Omron CX-Programmer project 新工程 (CX-Programmer 9.61)

# PLC 后氦检2: CJ2M CPU33
I/O table (CPU CJ2M-CPU33): rack 0 slot 0 CJ1W-SCU21-V1; rack 0 slot 1 CJ1W-AD041-V1; rack 0 slot 2 CJ1W-ID261; rack 0 slot 3 CJ1W-OD231; rack 0 slot 4 CJ1W-OC201; rack 0 slot 11 CJ2M-EIP21

## Global symbols (name address type ; comment)
0.00 BOOL  ; 外来拉有料感应1
0.01 BOOL  ; 上料有料感应
0.02 BOOL  ; 电池跟随检测
0.03 BOOL  ; 扫码位有料感应
0.04 BOOL  ; 上料位柔性报警（常闭）
0.05 BOOL  ; 上料提升气缸原位
0.06 BOOL  ; 上料提升气缸到位
0.07 BOOL  ; 上料升降气缸原位
0.08 BOOL  ; 上料升降气缸到位(右）
0.09 BOOL  ; 右升降缸原位
0.10 BOOL  ; 右升降缸到位
0.11 BOOL  ; 上料左夹爪张开位
0.12 BOOL  ; 上料左夹爪夹紧位
0.13 BOOL  ; 上料右夹爪张开位
0.14 BOOL  ; 上料右夹爪夹紧位
0.15 BOOL  ; #1氦检阀原位
100.04 BOOL  ; 报警清除
101.00 BOOL  ; 手动放料限制条件
101.01 BOOL  ; 上料手动放料条件
102.00 BOOL  ; 放料停止拉带
110.00 BOOL  ; 整机复位按钮(T)
11.05 BOOL  ; #1腔体氦检阀
12.00 BOOL  ; #2腔体氦检阀
12.11 BOOL  ; #3腔体氦检阀
131.04 BOOL  ; 左扫码(M)
13.06 BOOL  ; #4腔体氦检阀
1534.15 BOOL  ; 单元1的串口1协议宏执行标志
1544.15 BOOL  ; 单元1串口2协议执行标志
1550.03 BOOL  ; 单元2串口1异常退出
1559.15 BOOL  ; 单元2串口1协议宏执行标志
1584.15 BOOL  ; SCU21_3 Port#1 Protocol Macro Executing Flag
15.05 BOOL  ; --
1600.03 BOOL  ; SCU21_4 Port#1 Abort Switch
1609.15 BOOL  ; SCU21_4 Port#1 Protocol Macro Executing Flag
16.00 BOOL  ; 故障计时按钮
16.01 BOOL  ; 故障计时清空按钮
1.00 BOOL  ; #2氦检阀原位
1.01 BOOL  ; 氦检1合模气缸原位
1.02 BOOL  ; 氦检1合模气缸到位
1.03 BOOL  ; 氦检2合模气缸原位
1.04 BOOL  ; 氦检2合模气缸到位
1.05 BOOL  ; 下料提升气缸原位
1.06 BOOL  ; 下料提升气缸到位
1.07 BOOL  ; 进料扫码阻挡缩回
1.08 BOOL  ; 进料扫码阻挡伸出
1.09 BOOL  ; 下料左夹爪张开位
1.10 BOOL  ; 下料左夹爪夹紧位
1.11 BOOL  ; 下料右夹爪张开位
1.12 BOOL  ; 下料右夹爪夹紧位
1.13 BOOL  ; 可出料信号
1.14 BOOL  ; 内部机台对接（下机台输出信号7.01）
1.15 BOOL  ; 下料位有料感应3
2000 CHANNEL  ; #1真空计度读出值CHO
2001 CHANNEL  ; #1真空计读出值CH1
2002 CHANNEL  ; #2真空计读出值CH2
2029.00 BOOL  ; #1真空计断线
2029.01 BOOL  ; #2真空计断线
20.00 BOOL  ; 自动模式切换按钮(T)
20.01 BOOL  ; 自动启动按钮(T)
20.02 BOOL  ; 自动停止按钮(T)
20.06 BOOL  ; 氦检仪内部校准
20.07 BOOL  ; 柔性报警解除按钮(T)
20.12 BOOL  ; 氦检仪内部校准
2906.06 BOOL  ; 进料机械手左极限
2906.07 BOOL  ; 进料机械手右极限
2906.08 BOOL  ; 出料机械手左极限
2906.09 BOOL  ; 出料机械手右极限
2960.00 BOOL  ; 上料伺服原点
2960.01 BOOL  ; 上料伺服近原点
2960.02 BOOL  ; 下料伺服原点
2960.03 BOOL  ; 下料伺服近原点
2960.04 BOOL  ; 备用
2960.05 BOOL  ; 备用
2960.06 BOOL  ; 上料伺负向限位
2960.07 BOOL  ; 上料伺服正向限位
2960.08 BOOL  ; 下料伺服负方向限位
2960.09 BOOL  ; 下料伺服正方向限位
2961.00 BOOL  ; 上料伺服脉冲
2961.01 BOOL  ; 下料伺服脉冲
2961.02 BOOL  ; 上料伺服方向
2961.03 BOOL  ; 下料伺服方向
2961.04 BOOL  ; 下一机台故障时，控制下一机台出料输送带（接到下一台机的7.15同一电机）
2.00 BOOL  ; 氦检仪报警信号
2.01 BOOL  ; 内部机台对接信号（后面一台后氦检下料位有料感应，即3。01）
2.02 BOOL  ; 内部机台对接（后面一台后氦检的出料拉带末端有料感应，即3.03）
2.03 BOOL  ; 下料柔性报警（常闭）
2.04 BOOL  ; 气源压力信号
2.05 BOOL  ; 上料伺服准备好
2.06 BOOL  ; 下料伺服准备好
2.07 BOOL  ; 上料伺服报警
2.08 BOOL  ; 下料伺服报警
2.09 BOOL  ; NG气缸原位
2.10 BOOL  ; NG气缸到位
2.11 BOOL  ; 扫码NG缸原位
2.12 BOOL  ; 扫码NG缸到位
2.13 BOOL  ; 扫码NG放料位有料感应
2.14 BOOL  ; 扫码NG槽溢出
2.15 BOOL  ; 扫码NG放料位有料感应
31.04 BOOL  ; #1电池扫码按钮
3.00 BOOL  ; 下料位光栅感应(常闭)
3.01 BOOL  ; 腔体1有料
3.02 BOOL  ; 下料位有料感应(常闭)
3.03 BOOL  ; 下料拉带末端有料感应(常闭)
3.04 BOOL  ; NG溢出感应
3.05 BOOL  ; 真空泵缺相
3.06 BOOL  ; 腔体2有料
3.07 BOOL  ; 过渡拉带末端有料感应
3.08 BOOL  ; 启动按钮
3.09 BOOL  ; 停止按钮
3.10 BOOL  ; 复位按钮
3.11 BOOL  ; 急停按钮
3.12 BOOL  ; 前门禁信号
3.13 BOOL  ; 后门禁信号
3.14 BOOL  ; 左门禁信号
3.15 BOOL  ; 右门禁信号
52.00 BOOL  ; 全部清零按钮
52.02 BOOL  ; OK数清零按钮
52.04 BOOL  ; NG数清零按钮
6.00 BOOL  ; 上料提升气缸
6.01 BOOL  ; #1上料升降气缸（左）
6.02 BOOL  ; #2上料升降气缸（右）
6.03 BOOL  ; 上料左夹爪
6.04 BOOL  ; 上料右夹爪
6.05 BOOL  ; 氦检1合模气缸伸出 关腔体
6.06 BOOL  ; 氦检1合模气缸缩回 开腔体
6.07 BOOL  ; 氦检2合模气缸伸出
6.08 BOOL  ; 氦检2合模气缸缩回
6.09 BOOL  ; 氦检1抽真空阀
6.10 BOOL  ; 氦检1氦检阀
6.11 BOOL  ; 氦检1破真空阀
6.12 BOOL  ; 氦检1吹气阀
6.13 BOOL  ; 氦检2抽真空
6.14 BOOL  ; 氦检2氦检阀
6.15 BOOL  ; 氦检2破真空阀
782 CHANNEL  ; 校验通信异常延时
7.00 BOOL  ; 氦检2吹气阀
7.01 BOOL  ; 内部机台对接（本机台给上机台信号1.14）
7.02 BOOL  ; 扫码阻挡气缸
7.03 BOOL  ; 上料私服使能
7.04 BOOL  ; 下料私服使能
7.05 BOOL  ; 过渡拉带启动
7.06 BOOL  ; 氦检仪电源开启
7.07 BOOL  ; 氦检仪启动
7.08 BOOL  ; 下料提升气缸
7.09 BOOL  ; 上工站可往下放料信号
7.10 BOOL  ; 下料左夹爪
7.11 BOOL  ; 下料右夹爪
7.12 BOOL  ; NG气缸
7.13 BOOL  ; 扫码NG缸
7.14 BOOL  ; 进料输送带电机
7.15 BOOL  ; 出料输送带电机
8.00 BOOL  ; 启动指示灯
8.01 BOOL  ; 停止指示灯
8.02 BOOL  ; 复位指示灯
8.03 BOOL  ; 三色灯-红
8.04 BOOL  ; 三色灯-绿
8.05 BOOL  ; 三色灯-黄
8.06 BOOL  ; 蜂鸣器
8.07 BOOL  ; 真空泵
9.04 BOOL  ; 氦检电源打开
A202.01 BOOL  ; 通信端口1允许标志
A202.02 BOOL  ; 通信端口2允许标志
A202.03 BOOL  ; 通信端口3允许标志
A276 CHANNEL  ; 前机械手当前脉冲
A278 CHANNEL  ; 下料机械手当前脉冲
A280.04 BOOL  ; 上料机械手脉冲输出中
A280.05 BOOL  ; 上料轴无原点标志
A281.04 BOOL  ; 下料机械手脉冲输出中
A281.05 BOOL  ; 下料轴无原点标志
A322 CHANNEL  ; 进料旋转当前位置脉冲
A324 CHANNEL  ; 出料旋转当前位置脉冲
A326.04 BOOL  ; 进料旋转脉冲输出中
A326.05 BOOL  ; 上料旋转原点标志
A327.04 BOOL  ; 出料旋转脉冲输出中
A327.05 BOOL  ; 下料旋转原点标志
A351 CHANNEL  ; 系统时间
A540.08 BOOL  ; 上料机械手CW
A540.09 BOOL  ; 上料机械手CCW
A541.08 BOOL  ; 下料机械手CW
A541.09 BOOL  ; 下料机械手CCW
A542.08 BOOL  ; 进料旋转CCW
A542.09 BOOL  ; 进料旋转CW
A543.08 BOOL  ; 出料旋转CCW
A543.09 BOOL  ; 出料旋转CW
D0 CHANNEL  ; 上料机械手自动速度mm/s
D10 CHANNEL  ; 上料左夹位
D100 CHANNEL  ; 外来拉有料感应1延时HMI
D1000 CHANNEL  ; #1腔体检漏口压力(浮点)
D1002 CHANNEL  ; #1腔体漏率(浮点)
D1004 CHANNEL  ; #1腔体测试完成时的检漏口压力
D1006 CHANNEL  ; #1腔体测试完成时的漏率
D101 CHANNEL  ; 外来拉有料感应2延时HMI
D102 CHANNEL  ; 上料位有料感应延时HMI
D1020 CHANNEL  ; #2腔体检漏口压力(浮点)
D1022 CHANNEL  ; #2腔体漏率(浮点)
D1024 CHANNEL  ; #2腔体测试完成时检漏口压力
D1026 CHANNEL  ; #2腔体测试完成时的漏率
D103 CHANNEL  ; 上料位有料感应2延时HMI
D104 CHANNEL  ; 上料位柔性报警（常闭）延时
D105 CHANNEL  ; 上料提升气缸原位延时
D106 CHANNEL  ; 上料提升气缸到位延时
D107 CHANNEL  ; 上料升降气缸原位延时
D108 CHANNEL  ; 上料升降气缸到位延时
D109 CHANNEL  ; 扫码阻挡气缸原位延时
D110 CHANNEL  ; 扫码阻挡气缸到位延时
D1100 CHANNEL  ; 测试
D111 CHANNEL  ; 上料左夹爪张开位延时
D112 CHANNEL  ; 上料左夹爪夹紧位延时
D113 CHANNEL  ; 上料右夹爪张开位延时
D114 CHANNEL  ; 上料右夹爪夹紧位延时
D1140 CHANNEL  ; HMI 页面
D115 CHANNEL  ; #1氦检阀原位延时时间
D116 CHANNEL  ; #2氦检阀原位延时时间
D117 CHANNEL  ; 氦检1合模气缸原位延时
D118 CHANNEL  ; 氦检1合模气缸到位延时
D119 CHANNEL  ; 氦检2合模气缸原位延时
D12 CHANNEL  ; 下料右夹爪OK放料位
D120 CHANNEL  ; 氦检2合模气缸到位延时
D1204 CHANNEL  ; 检漏口压力设定值
D1206 CHANNEL  ; 漏率设定值
D121 CHANNEL  ; 下料提升气缸原位延时
D1210 CHANNEL  ; 氦检仪稳定设定时间
D122 CHANNEL  ; 下料提升气缸到位延时
D123 CHANNEL  ; 下料升降气缸原位延时
D124 CHANNEL  ; 下料升降气缸到位延时
D125 CHANNEL  ; 下料左夹爪张开位延时
D1250 CHANNEL  ; 检漏口压力设定值小数部分
D1252 CHANNEL  ; 检漏口压力设定值指数
D1254 CHANNEL  ; 漏率设定值小数部分
D1256 CHANNEL  ; 漏率设定值指数
D126 CHANNEL  ; 下料左夹爪夹紧位延时
D1260 CHANNEL  ; 检漏口压力底数转换
D1264 CHANNEL  ; 漏率底数转换
D1266 CHANNEL  ; 漏率设定值(浮点数Pa.m3)
D127 CHANNEL  ; 下料右夹爪张开位延时
D1270 CHANNEL  ; 注氦嘴气密性设定值小数部分
D1272 CHANNEL  ; 注氦嘴气密性设定值指数
D1274 CHANNEL  ; 注氦嘴气密性设定值指数部分
D1276 CHANNEL  ; 注氦嘴气密性设定值(Float)
D1278 CHANNEL  ; 清氦次数设定值
D128 CHANNEL  ; 下料右夹爪夹紧位延时
D129 CHANNEL  ; 备用
D130 CHANNEL  ; 备用
D131 CHANNEL  ; 备用
D1310 CHANNEL  ; 氦检仪稳定漏率设定值小数
D1312 CHANNEL  ; 氦检仪稳定漏率设定值指数
D1316 CHANNEL  ; 氦检仪稳定漏率设定值(Float)
D132 CHANNEL  ; 氦检仪报警信号延时
D133 CHANNEL  ; 备用
D134 CHANNEL  ; 备用
D135 CHANNEL  ; 下料柔性报警（常闭）延时
D136 CHANNEL  ; 气源压力信号延时
D137 CHANNEL  ; 上料伺服准备好延时
D138 CHANNEL  ; 下料伺服准备好延时
D139 CHANNEL  ; 备用
D140 CHANNEL  ; 备用
D141 CHANNEL  ; NG气缸原位延时
D1416 CHANNEL  ; 氦检仪压力异常延时
D142 CHANNEL  ; NG气缸到位延时
D143 CHANNEL  ; 工站给予信号时间
D144 CHANNEL  ; 扫码NG缸原位时间
D145 CHANNEL  ; 扫码NG缸原位时间
D146 CHANNEL  ; 备用
D147 CHANNEL  ; 备用
D148 CHANNEL  ; 1#腔体有料延时
D149 CHANNEL  ; 2#腔体有料延时
D150 CHANNEL  ; 下料位有料感应1延时
D151 CHANNEL  ; 下料位有料感应2延时
D152 CHANNEL  ; NG溢出感应延时
D153 CHANNEL  ; 真空泵缺相延时
D154 CHANNEL  ; 备用
D155 CHANNEL  ; 备用
D156 CHANNEL  ; 启动按钮延时
D157 CHANNEL  ; 停止按钮延时
D158 CHANNEL  ; 复位按钮延时
D159 CHANNEL  ; 急停按钮延时
D1590 CHANNEL  ; 扫码位暂存码1
D16 CHANNEL  ; 上料左扫码NG参数
D160 CHANNEL  ; 前门禁信号延时
D1600 CHANNEL  ; 扫码位暂存码
D161 CHANNEL  ; 后门禁信号延时
D162 CHANNEL  ; 左门禁信号延时
D163 CHANNEL  ; 右门禁信号延时
D168 CHANNEL  ; 传感器延迟时间
D1790 CHANNEL  ; 上料位待料延时设定HMI
D18 CHANNEL  ; 上料右扫码NG参数
D180 CHANNEL  ; 上料机械手当前脉冲
D1802 CHANNEL  ; TS
D182 CHANNEL  ; 上料机械手当前脉冲(浮点)
D184 CHANNEL  ; 伺服脉冲当量(浮点)
D1840 CHANNEL  ; 下料右爪测试检漏口压力结果
D1842 CHANNEL  ; 下料右爪测试漏率结果
D1844 CHANNEL  ; 下料右爪 测试结果
D1846 CHANNEL  ; 下料左爪压力
D1848 CHANNEL  ; 下料左爪漏率
D1850 CHANNEL  ; 下料左爪测试结果
D1858 CHANNEL  ; 下料右爪测试检漏口压力结果PC
D186 CHANNEL  ; 上料机械手当前位置(mm)
D1860 CHANNEL  ; 下料右爪测试漏率结果PC
D1862 CHANNEL  ; 下料右爪 测试结果pC
D1868 CHANNEL  ; 下料左爪压力PC
D1870 CHANNEL  ; 下料左爪漏率PC
D1872 CHANNEL  ; 下料左爪测试结果PC
D188 CHANNEL  ; 伺服脉冲当量
D1880 CHANNEL  ; 1爪腔体编号
D1881 CHANNEL  ; 2爪腔体编号
D190 CHANNEL  ; 下料机械手当前脉冲
D1900 CHANNEL  ; 下料右爪电池工位PC
D1901 CHANNEL  ; 传输完成地址
D1902 CHANNEL  ; 下料左爪工位PC
D1903 CHANNEL  ; 传输完成-左
D1904 CHANNEL  ; 传输完成地址
D1905 CHANNEL  ; 传输完成-左
D192 CHANNEL  ; 下料机械手当前脉冲(浮点)
D196 CHANNEL  ; 下料机械手当前位置(mm)
D198 CHANNEL  ; 上下料机械手距各自原点的总距离
D2 CHANNEL  ; 上料机械手手动速度mm/s
D20 CHANNEL  ; 下料机械手自动速度mm/s
D200 CHANNEL  ; #1腔体真空值
D2000 CHANNEL  ; 氦检仪当前实时漏率
D20000 CHANNEL  ; #1,#2路模拟量使用设置
D20001 CHANNEL  ; #1,#2路模拟量输入范围位0--10v
D20018 CHANNEL  ; #1,#2路模拟量分辨率8000，普通模式
D210 CHANNEL  ; #2腔体真空值
D22 CHANNEL  ; 下料机械手动速度mm/s
D230 CHANNEL  ; #1腔体抽气时间
D232 CHANNEL  ; #2腔体抽气时间
D234 CHANNEL  ; 1屏蔽2带料3测试中4测试完成
D236 CHANNEL  ; 1屏蔽2带料3测试中4测试完成
D238 CHANNEL  ; #1腔体测试结果
D239 CHANNEL  ; #2腔体测试结果
D24 CHANNEL  ; 下料机械手腔体1位置(mm)
D240 CHANNEL  ; 接收检漏仪状态的起始字
D241 CHANNEL  ; 接收的检漏口压力(ASCII)
D2450 CHANNEL  ; 氦捡仪稳定时间设定值(BCD)
D2452 CHANNEL  ; #1氦检阀打开抽气阀关闭延时
D2454 CHANNEL  ; #2氦检阀打开抽气阀关闭延时
D2456 CHANNEL  ; 氦检关真空延时
D250 CHANNEL  ; 接收检漏口压力的起始字
D251 CHANNEL  ; 接收的检漏口压力(ASCII)
D26 CHANNEL  ; 下料机械手腔体2位置(mm)
D260 CHANNEL  ; 接收漏率起始字
D261 CHANNEL  ; 接收的漏率(ASCII)
D270 CHANNEL  ; 上下料机械手原点间距离
D272 CHANNEL  ; 机械手治具宽度
D274 CHANNEL  ; 上下料机械手间的距离
D28 CHANNEL  ; 下料机械手左夹爪OK放料位置(mm)
D282 CHANNEL  ; .
D290 CHANNEL  ; 180浮点数
D294 CHANNEL  ; 180度脉冲数
D298 CHANNEL  ; 进料位置+180度角
D30 CHANNEL  ; 下料机械手NG放料位置(mm)
D300 CHANNEL  ; 外来拉有料感应1延时
D301 CHANNEL  ; 外来料感应2
D302 CHANNEL  ; 上料位有料感应1
D303 CHANNEL  ; 上料位有料延时
D304 CHANNEL  ; 柔性报警
D3040 CHANNEL  ; 取料位条码
D305 CHANNEL  ; 上料提升原位延时
D306 CHANNEL  ; 上料提升延时
D3060 CHANNEL  ; 右夹子条码
D307 CHANNEL  ; 上料升降延时
D308 CHANNEL  ; 上料升降到位延时
D3080 CHANNEL  ; 上料左夹子条码
D309 CHANNEL  ; 右升降原位延时间
D310 CHANNEL  ; 右升降缸到位时间
D3100 CHANNEL  ; 腔体1右待测料条码
D311 CHANNEL  ; 上左爪张开位
D312 CHANNEL  ; 上左夹紧延时
D3120 CHANNEL  ; 腔体2左位条码
D313 CHANNEL  ; 上右爪松开延时
D314 CHANNEL  ; 上右夹紧延时
D3140 CHANNEL  ; 腔体2右位条码
D3160 CHANNEL  ; 腔体1左待测条码
D317 CHANNEL  ; 合模1原位延时
D318 CHANNEL  ; 合模1到位延时
D3180 CHANNEL  ; 下料右爪条码
D319 CHANNEL  ; 合模2原位延时
D32 CHANNEL  ; 出料旋转步进自动速度(度/s）
D320 CHANNEL  ; 合模2到位延时
D3200 CHANNEL  ; 下料左爪条码
D321 CHANNEL  ; 下料提升原位延时
D322 CHANNEL  ; 下料提升到位延时
D3220 CHANNEL  ; 下料右爪条码PC
D323 CHANNEL  ; 备用
D324 CHANNEL  ; 备用
D3240 CHANNEL  ; 下料左爪条码PC
D325 CHANNEL  ; 下左爪张开延时
D326 CHANNEL  ; 下左夹紧延时
D327 CHANNEL  ; 下右爪张开位延时
D328 CHANNEL  ; 下右爪夹紧位延时
D332 CHANNEL  ; 氦检报警延时
D335 CHANNEL  ; 下料柔性报警延时
D336 CHANNEL  ; 气压报警延时
D34 CHANNEL  ; 出料旋转步进手动速度(度/s)
D341 CHANNEL  ; NG气缸原位延时
D342 CHANNEL  ; NG气缸到位延时
D348 CHANNEL  ; 1#腔体有料延时
D349 CHANNEL  ; 2#腔体有料延时
D350 CHANNEL  ; 下料位有料感应1延时
D351 CHANNEL  ; 下料位有料感应2延时
D353 CHANNEL  ; 真空泵缺相
D36 CHANNEL  ; 出料旋转步进出料角度1(mm)
D370 CHANNEL  ; 氦检仪就绪状态
D38 CHANNEL  ; 出料旋转步进下料角度
D4 CHANNEL  ; 上料机械手右夹爪位(浮点)
D40 CHANNEL  ; 腔体真空达到阀值
D400 CHANNEL  ; 上料机械手自动状态加速度
D4000 CHANNEL  ; 真空值1转存
D4002 CHANNEL  ; #1真空值运算1
D4004 CHANNEL  ; #1真空值运算2
D4006 CHANNEL  ; #1真空值运算3
D4008 CHANNEL  ; #1真空值运算4
D401 CHANNEL  ; 上料机械手自动状态减速度
D4010 CHANNEL  ; 腔体1实际真空值(浮点)
D402 CHANNEL  ; 上料机械手自动速度puls/s
D4020 CHANNEL  ; 真空值2转存
D4022 CHANNEL  ; #2真空值运算1
D4024 CHANNEL  ; #2真空值运算2
D4026 CHANNEL  ; #2真空值运算3
D4028 CHANNEL  ; #2真空值运算4
D404 CHANNEL  ; 上料机械手自动位移量
D406 CHANNEL  ; 上料机械手自动状态起动速度
D410 CHANNEL  ; 上料机械手手动状态加速度
D411 CHANNEL  ; 上料机械手手动状态减速度
D412 CHANNEL  ; 上料机械手手动速度puls/s
D414 CHANNEL  ; 上料机械手手动位移量
D416 CHANNEL  ; 上料机械手手动状态起动速度
D42 CHANNEL  ; 腔体抽气时间
D420 CHANNEL  ; 下料机械手自动状态加速度
D421 CHANNEL  ; 下料机械手自动状态减速度
D422 CHANNEL  ; 下料机械手自动速度puls/s
D424 CHANNEL  ; 下料机械手自动位移量
D426 CHANNEL  ; 下料机械手自动状体起动速度
D430 CHANNEL  ; 下料机械手手动状态加速度
D431 CHANNEL  ; 下料机械手手动状态减速度
D432 CHANNEL  ; 下料机械手手动速度puls/s
D434 CHANNEL  ; 下料机械手手动位移量
D436 CHANNEL  ; 下料机械手手动状态起动速度
D44 CHANNEL  ; 抽残气后压力设置值
D440 CHANNEL  ; 进料旋转步进自动状态加速度
D441 CHANNEL  ; 进料旋转步进自动状体减速度
D442 CHANNEL  ; 进料旋转步进自动速度puls/s
D444 CHANNEL  ; 进料旋转自动位移量
D446 CHANNEL  ; 进料旋转步进自动状态起动速度
D450 CHANNEL  ; 进料旋转步进手动状态加速度
D451 CHANNEL  ; 进料旋转步进手动状态减速度
D452 CHANNEL  ; 进料旋转步进手动速度puls/s
D456 CHANNEL  ; 进料旋转步进手动状态起动速度
D46 CHANNEL  ; 氦检设定时间
D460 CHANNEL  ; 出料旋转步进自动状态加速度
D461 CHANNEL  ; 出料旋转步进自动状态减速度
D462 CHANNEL  ; 出料旋转步进自动速度puls/s
D464 CHANNEL  ; 出料旋转自动位移量
D466 CHANNEL  ; 出料旋转步进自动状态起动速度
D470 CHANNEL  ; 出料旋转步进手动状态加速度
D471 CHANNEL  ; 出料旋转步进手动状态减速度
D472 CHANNEL  ; 出料旋转步进手动速度puls/s
D476 CHANNEL  ; 出料旋转步进手动状态起动速度
D48 CHANNEL  ; 腔体破真空设定值
D480 CHANNEL  ; 上下料机械手正向行程脉冲
D484 CHANNEL  ; 上下料机械手反向行程
D488 CHANNEL  ; 上下料机械手反向行程脉冲
D50 CHANNEL  ; 检漏口压力指数
D500 CHANNEL  ; 上料机械手自动速度puls/s
D5000 CHANNEL  ; 扫码1长度
D504 CHANNEL  ; 上料机械手手动速度puls/s
D510 CHANNEL  ; 下料机械手自动速度puls/s
D514 CHANNEL  ; 下料机械手手动速度puls/s
D5198 CHANNEL  ; 流入个数
D52 CHANNEL  ; 检漏口压力底数
D520 CHANNEL  ; 进料旋转步进自动速度puls/s
D5200 CHANNEL  ; 流出个数
D5202 CHANNEL  ; OK个数
D5204 CHANNEL  ; 检测NG个数
D5206 CHANNEL  ; 良率
D5220 CHANNEL  ; 扫码NG个数
D5222 CHANNEL  ; 检测产量
D524 CHANNEL  ; 进料旋转步进手动速度puls/s
D530 CHANNEL  ; 出料旋转步进自动速度puls/s
D534 CHANNEL  ; 出料旋转步进手动速度puls/s
D54 CHANNEL  ; 漏率指数
D5430 CHANNEL  ; PPM统计
D5432 CHANNEL  ; 下料数量
D5434 CHANNEL  ; 计时
D550 CHANNEL  ; 上料机械手在（右）扫码NG位..
D552 CHANNEL  ; 上料机械手在（左）NG槽参数
D56 CHANNEL  ; 漏率底数
D580 CHANNEL  ; 下料右爪放OK料位置（浮点）
D584 CHANNEL  ; 下料右爪放OK料位置脉冲
D592 CHANNEL  ; 上料机械手左夹爪位置脉冲(浮点)
D596 CHANNEL  ; 上料机械手左夹爪位置脉冲
D6 CHANNEL  ; 上料机械手腔体1位置(浮点)
D60 CHANNEL  ; 腔体自检真空阀值
D600 CHANNEL  ; 上料机械手右夹爪位置脉冲(浮点)
D602 CHANNEL  ; 氦检上限位值
D604 CHANNEL  ; 上料机械手右夹爪位置脉冲
D610 CHANNEL  ; 上料机械手腔体1位置脉冲(浮点)
D6100 CHANNEL  ; 2个电芯出料计时
D614 CHANNEL  ; 上料机械手腔体1位置脉冲
D62 CHANNEL  ; 腔体自检抽气时间
D620 CHANNEL  ; 上料机械手腔体2位置(浮点)
D6200 CHANNEL  ; 2个电芯生产周期
D624 CHANNEL  ; 上料机械手腔体2位置脉冲
D626 CHANNEL  ; 上料机械手在（右）扫码NG位
D628 CHANNEL  ; 上料机械手在（左）NG槽参数
D630 CHANNEL  ; 下料机械手腔体1位置(浮点)
D6300 CHANNEL  ; PPM
D634 CHANNEL  ; 下料机械手腔体1位置脉冲
D64 CHANNEL  ; 腔体自检泄漏量设置值
D640 CHANNEL  ; 下料机械手腔体2位置(浮点)
D644 CHANNEL  ; 下料机械手腔体2位置脉冲
D650 CHANNEL  ; 下料机械手左爪OK放料位置(浮点)
D654 CHANNEL  ; 下料机械手左爪OK放料位置脉冲
D66 CHANNEL  ; 条码设置长度
D660 CHANNEL  ; 下料机械手NG放料位置(浮点)
D664 CHANNEL  ; 下料机械手NG放料位置脉冲
D670 CHANNEL  ; 氦检下限位值
D672 CHANNEL  ; 氦检上限位值
D674 CHANNEL  ; 进料旋转进料位置1脉冲
D68 CHANNEL  ; 腔体自检保压前设定时间
D680 CHANNEL  ; 进料旋转上料位置(浮点)
D684 CHANNEL  ; 进料旋转上料位置脉冲
D688 CHANNEL  ; 进料旋转上料位置+180度位置脉冲
D690 CHANNEL  ; 出料旋转出料位置1(浮点)
D694 CHANNEL  ; 出料旋转出料位置1脉冲
D70 CHANNEL  ; 腔体自检保压设定时间
D700 CHANNEL  ; 出料旋转下料位置(浮点)
D7000 CHANNEL  ; #1扫码长度
D7001 CHANNEL  ; #1电池条码
D704 CHANNEL  ; 出料旋转下料位置脉冲
D710 CHANNEL  ; 旋转步进正向行程脉冲
D714 CHANNEL  ; 旋转步进反向行程
D72 CHANNEL  ; 腔体自检破真空设定值
D720 CHANNEL  ; 轴控制预留
D734 CHANNEL  ; 旋转步进反向行程脉冲
D74 CHANNEL  ; #1腔体保压前真空值
D76 CHANNEL  ; #1腔体保压后真空值
D78 CHANNEL  ; #1腔体自检泄漏量
D780 CHANNEL  ; 进料旋转步进进料角度2(mm)
D782 CHANNEL  ; 进料旋转进料位置2(浮点)
D784 CHANNEL  ; 进料旋转进料位置2脉冲
D792 CHANNEL  ; 出料旋转出料位置2(浮点)
D794 CHANNEL  ; 出料旋转出料位置2脉冲
D8 CHANNEL  ; 上料机械手腔体2位置(浮点)
D80 CHANNEL  ; #2腔体保压前真空值
D800 CHANNEL  ; 氦检时间(储存)
D8000 CHANNEL  ; 检漏状态第一字节
D8001 CHANNEL  ; 检漏状态第二字节
D8002 CHANNEL  ; 检漏状态结束字节
D8010 CHANNEL  ; 待机状态第一字节
D8011 CHANNEL  ; 待机状态第二字节
D8012 CHANNEL  ; 待机状态结束字节
D802 CHANNEL  ; 检漏口压力指数(储存)
D8020 CHANNEL  ; 定标状态第一字节
D8021 CHANNEL  ; 定标状态第二字节
D8022 CHANNEL  ; 定标状态结束字节
D8030 CHANNEL  ; 启动状态第一字节
D8031 CHANNEL  ; 启动状态第二字节
D8032 CHANNEL  ; 启动状态结束字节
D804 CHANNEL  ; 检漏口压力底数(储存)
D8040 CHANNEL  ; 错误状态第一字节
D8041 CHANNEL  ; 错误状态第二字节
D8042 CHANNEL  ; 错误状态结束字节
D8050 CHANNEL  ; 暂停状态第一字节
D8051 CHANNEL  ; 暂停状态第二字节
D8052 CHANNEL  ; 暂停状态结束字节
D806 CHANNEL  ; 漏率指数
D808 CHANNEL  ; 漏率底数
D8100 CHANNEL  ; 氦检仪状态(1-检漏,2-待机,3-启动,4-定标,5-错误,6-暂停)
D82 CHANNEL  ; #1腔体保压后真空值
D820 CHANNEL  ; 设备状态
D821 CHANNEL  ; 设备状态(储存)
D822 CHANNEL  ; 设备状态变更
D830 CHANNEL  ; 早班分、秒
D8300 CHANNEL  ; 校验触发
D8302 CHANNEL  ; 校验结果（1-OK，2-NG）
D831 CHANNEL  ; 早班日、时
D832 CHANNEL  ; 晚班分、秒
D833 CHANNEL  ; 晚班分、秒
D834 CHANNEL  ; 晚班日、时
D836 CHANNEL  ; 只比较时、分、秒
D838 CHANNEL  ; 晚班传输信号
D84 CHANNEL  ; #2腔体自检泄漏量
D840 CHANNEL  ; 单班生产时间
D8400 CHANNEL  ; 读氦检仪报警
D842 CHANNEL  ; 单班故障时间
D8500 CHANNEL  ; 读氦检仪内部校准状态
D8600 CHANNEL  ; 氦检校准暂存状态1-完成
D8601 CHANNEL  ; 氦检校准暂存状态1-完成
D8610 CHANNEL  ; 氦检校准暂存状态2-通过
D8611 CHANNEL  ; 氦检校准暂存状态2-通过
D8612 CHANNEL  ; 氦检校准暂存状态3
D8620 CHANNEL  ; 氦检校准暂存状态3-进行
D8621 CHANNEL  ; 氦检校准暂存状态3-进行
D8622 CHANNEL  ; 氦检校准暂存状态3-进行
D90 CHANNEL  ; #1腔体手动抽气时间
D9000 CHANNEL  ; PC交换地址
D91 CHANNEL  ; #1腔体保压前时间
D9100 CHANNEL  ; 上下料机械手总距离
D9102 CHANNEL  ; 原点距离
D9104 CHANNEL  ; 2轴相距距离
D92 CHANNEL  ; #1腔体保压时间
D93 CHANNEL  ; #2腔体自检抽气时间
D9300 CHANNEL  ; 放料状态
D94 CHANNEL  ; #2腔体进入保压前时间
D95 CHANNEL  ; #2腔体保压时间
D9500 CHANNEL  ; #1放料电池条码
D9520 CHANNEL  ; #2放料电池条码
D9591 CHANNEL  ; #1放料电池条码
D9592 CHANNEL  ; #1放料电池条码
D9593 CHANNEL  ; #1放料电池条码
D9594 CHANNEL  ; #1放料电池条码
D9595 CHANNEL  ; #1放料电池条码
D9596 CHANNEL  ; #1放料电池条码
D9597 CHANNEL  ; #1放料电池条码
D9598 CHANNEL  ; #1放料电池条码
D9599 CHANNEL  ; #1放料电池条码
D9601 CHANNEL  ; #2放料电池条码
D9602 CHANNEL  ; #2放料电池条码
D9603 CHANNEL  ; #2放料电池条码
D9604 CHANNEL  ; #2放料电池条码
D9605 CHANNEL  ; #2放料电池条码
D9606 CHANNEL  ; #2放料电池条码
D9607 CHANNEL  ; #2放料电池条码
D9608 CHANNEL  ; #2放料电池条码
D9609 CHANNEL  ; #2放料电池条码
D9612 CHANNEL  ; 放料电池实际漏率
D9613 CHANNEL  ; 放料电池实际漏率
D9614 CHANNEL  ; 放料电池实际检漏口压力
D9615 CHANNEL  ; 放料电池实际检漏口压力
D9616 CHANNEL  ; 放料电池电池工位
D9617 CHANNEL  ; 放料电池电池工位
D9618 CHANNEL  ; 放料电池电池测试结果
D9619 CHANNEL  ; 放料电池电池测试结果
D9630 CHANNEL  ; 漏率设定值
D9631 CHANNEL  ; 漏率设定值
D9632 CHANNEL  ; 检漏口压力设定值
D9633 CHANNEL  ; 检漏口压力设定值
D9634 CHANNEL  ; 氦检时间设定值
D9635 CHANNEL  ; 氦检时间设定值
D9999 CHANNEL  ; 程序修改日期
H0.00 BOOL  ; #1腔体启用
H0.01 BOOL  ; #2腔体启用
H0.02 BOOL  ; 扫码屏蔽（1-屏蔽)
H0.03 BOOL  ; 电脑屏蔽
H0.04 BOOL  ; 门磁开关启用
H0.05 BOOL  ; 0-正常程序/1-空跑程序
H0.06 BOOL  ; 氦检仪屏蔽
H0.07 BOOL  ; 重复扫码禁用
H0.08 BOOL  ; 真空屏蔽
H0.09 BOOL  ; 入料拉带停止选择
H10.00 BOOL  ; 夹爪下料区有电池
H110.00 BOOL  ; 新复位方式启用
H11.00 BOOL  ; 上料机械手归零完成
H16.02 BOOL  ; 下料夹爪1手动松开
H16.03 BOOL  ; 下料夹爪2手动松开
H16.04 BOOL  ; 下料夹爪3手动松开
H16.05 BOOL  ; 下料夹爪4手动松开
H1.00 BOOL  ; 外来拉有料感应1
H1.01 BOOL  ; 外来拉有料感应2(备用)
H1.02 BOOL  ; 上料位有料感应1
H1.03 BOOL  ; 上料位有料感应2
H1.04 BOOL  ; 上料位柔性报警（常闭）
H1.05 BOOL  ; 上料提升气缸原位
H1.06 BOOL  ; 上料提升气缸到位
H1.07 BOOL  ; 上料升降气缸原位
H1.08 BOOL  ; 上料升降气缸到位
H1.09 BOOL  ; 右升降缸原位屏蔽
H1.10 BOOL  ; 右升降缸到位屏蔽
H1.11 BOOL  ; 上料左夹爪张开位
H1.12 BOOL  ; 上料左夹爪夹紧位
H1.13 BOOL  ; 上料右夹爪张开位
H1.14 BOOL  ; 上料右夹爪夹紧位
H1.15 BOOL  ; #1氦检阀原位屏蔽
H2.00 BOOL  ; #2氦检阀原位屏蔽
H2.01 BOOL  ; 氦检1合模气缸原位
H2.02 BOOL  ; 氦检1合模气缸到位
H2.03 BOOL  ; 氦检2合模气缸原位
H2.04 BOOL  ; 氦检2合模气缸到位
H2.05 BOOL  ; 下料提升气缸原位
H2.06 BOOL  ; 下料提升气缸到位
H2.07 BOOL  ; 备用
H2.08 BOOL  ; 备用
H2.09 BOOL  ; 下料左夹爪张开位
H2.10 BOOL  ; 下料左夹爪夹紧位
H2.11 BOOL  ; 下料右夹爪张开位
H2.12 BOOL  ; 下料右夹爪夹紧位
H2.13 BOOL  ; 备用
H2.14 BOOL  ; 备用
H2.15 BOOL  ; 备用
H3.00 BOOL  ; 氦检仪报警信号
H3.01 BOOL  ; 备用
H3.02 BOOL  ; 备用
H3.03 BOOL  ; 下料柔性报警（常闭）
H3.04 BOOL  ; 气源压力信号
H3.05 BOOL  ; 上料伺服准备好
H3.06 BOOL  ; 下料伺服准备好
H3.07 BOOL  ; 备用
H3.08 BOOL  ; 备用
H3.09 BOOL  ; NG气缸原位
H3.10 BOOL  ; NG气缸到位
H3.11 BOOL  ; 下个工站给予信号
H3.12 BOOL  ; 扫码NG气缸原位屏蔽
H3.13 BOOL  ; 扫码NG气缸到位屏蔽
H3.14 BOOL  ; 备用
H3.15 BOOL  ; 备用
H40.02 BOOL  ; 扫码屏蔽-HMI
H40.07 BOOL  ; 扫码NG料（右）
H40.08 BOOL  ; 扫码NG（左）
H46.00 BOOL  ; 机台方向选择(0:左进右出,1:右进左出)
H4.00 BOOL  ; 1#腔体有料
H4.01 BOOL  ; 2#腔体有料
H4.02 BOOL  ; 下料位有料感应1
H4.03 BOOL  ; 下料位有料感应2
H4.04 BOOL  ; NG溢出感应
H4.05 BOOL  ; 真空泵缺相
H4.06 BOOL  ; 备用
H4.07 BOOL  ; 备用
H4.08 BOOL  ; 启动按钮
H4.09 BOOL  ; 停止按钮
H4.10 BOOL  ; 复位按钮
H4.11 BOOL  ; 急停按钮
H4.12 BOOL  ; 前门禁信号
H4.13 BOOL  ; 后门禁信号
H4.14 BOOL  ; 左门禁信号
H4.15 BOOL  ; 右门禁信号
H50 CHANNEL  ; 复位有料记忆
H50.00 BOOL  ; 扫码位有料
H50.01 BOOL  ; 上料左爪有料记忆
H50.02 BOOL  ; 上料右爪有料
H50.03 BOOL  ; 下料右爪有料
H50.04 BOOL  ; 下料右爪有料
H50.05 BOOL  ; 爪子无料
H50.06 BOOL  ; 上料位有料标志
H50.07 BOOL  ; 上右夹爪有料标志
H50.08 BOOL  ; 上左夹有料标志
H50.09 BOOL  ; #1腔体右位有待测料标志
H50.10 BOOL  ; #1腔体左位有料标志
H50.11 BOOL  ; 2号腔体右位有料标志
H50.12 BOOL  ; 2#腔体左位有料标志
H50.13 BOOL  ; #1腔体NG
H50.14 BOOL  ; #1腔体测试中
H51.00 BOOL  ; #1腔体测试结束
H51.01 BOOL  ; #2腔体测试结束
H51.02 BOOL  ; 下料左爪有料
H51.03 BOOL  ; 下料右爪有料标志
H51.04 BOOL  ; #2腔体放料完成
H51.05 BOOL  ; 腔体1放料完成标志
H51.06 BOOL  ; #2腔体产品NG
H51.07 BOOL  ; #2腔体测试中
H51.13 BOOL  ; 去腔体#2取料标志
H51.14 BOOL  ; 下料轴往1#取料标志
H53.00 BOOL  ; 上料轴归零完成
H53.01 BOOL  ; #1腔体自检泄露
H53.02 BOOL  ; #2腔体自检泄露
H54.00 BOOL  ; 下料轴归零完成
H55.00 BOOL  ; 上料轴往1#腔体放料标志
H55.01 BOOL  ; 上料轴往2#腔体放料标志
H56.00 BOOL  ; 跟随检测
H5.00 BOOL  ; 氦检仪屏蔽
H5.02 BOOL  ; 蜂鸣器屏蔽
H5.09 BOOL  ; MES采集漏率单位为mPa.m3/s(仪器显示值1000倍)
H60.09 BOOL  ; #1腔体右位有待测料
H60.10 BOOL  ; #1腔体左位有料标志
H60.11 BOOL  ; 2号腔体右位有料
H60.12 BOOL  ; 2#腔体左位有料
H6.00 BOOL  ; 机台方向选择(0:左进右出,1:右进左出)
H80.00 BOOL  ; 左爪手动记忆有料
H80.01 BOOL  ; 右爪手动记忆有料
H80.02 BOOL  ; 上料左爪手动记忆有料
H80.03 BOOL  ; 上料右爪手动记忆有料
H80.05 BOOL  ; 下料拉带2有料
H80.06 BOOL  ; 过渡拉带有料
H81.00 BOOL  ; 老氦检仪选择
H81.01 BOOL  ; 氦检仪电源打开—HMI
H9.00 BOOL  ; 单料模式
T0000 BOOL  ; 进料感应延时
T0001 BOOL  ; 上料柔性报警感应延时
T0002 BOOL  ; 下料柔性报警感应延时
T0003 BOOL  ; 出料柔性报警感应延时
T0004 BOOL  ; 气源压力信号感应延时
T0005 BOOL  ; 进料缓存有料信号延时
T0006 BOOL  ; 出料缓存有料信号延时
T0007 BOOL  ; 腔体有料信号
T0008 BOOL  ; 扫码缓存左有料信号延时
T0009 BOOL  ; 扫码缓存右有料信号延时
T0010 BOOL  ; 右升降缸原位延时
T0011 BOOL  ; 右升降缸到位延时
T0014 BOOL  ; 上料左升降气缸缩回位时间
T0015 BOOL  ; 上料升降气缸伸出位延时
T0016 BOOL  ; 上料左夹爪张开位延时
T0017 BOOL  ; 上料夹爪1夹紧位延时
T0018 BOOL  ; 上料右爪张开位延时
T0019 BOOL  ; 上料右夹爪夹紧位延时
T0020 BOOL  ; 腔体1有料延时
T0021 BOOL  ; 腔体2有料
T0022 BOOL  ; 氦检仪稳定延时
T0023 BOOL  ; 氦检仪使用开始延时1s读取状态
T0028 BOOL  ; #2氦检阀原位延时
T0029 BOOL  ; #1氦检阀原位延时
T0030 BOOL  ; 合模气缸1原位延时
T0031 BOOL  ; 合模气缸1伸出位延时
T0032 BOOL  ; 合模气缸2原位延时
T0033 BOOL  ; 合模气缸2伸出位延时
T0034 BOOL  ; 下料提升气缸缩回位延时
T0035 BOOL  ; 下料提升气缸伸出位延时
T0036 BOOL  ; 下料左夹爪张开位延时
T0037 BOOL  ; 下料左爪夹紧位延时
T0038 BOOL  ; 下料右夹爪张开位延时
T0039 BOOL  ; 下料右爪2夹紧位延时
T0040 BOOL  ; 工站给予信号
T0041 BOOL  ; 扫码位没料延时
T0048 BOOL  ; 备用
T0049 BOOL  ; 备用
T0050 BOOL  ; 出料夹爪1张开位延时
T0051 BOOL  ; 出料夹爪1夹紧位延时
T0052 BOOL  ; 出料夹爪2张开位延时
T0053 BOOL  ; 出料夹爪2夹紧位延时
T0054 BOOL  ; 出料移栽气缸缩回位延时
T0055 BOOL  ; 出料移栽气缸伸出位延时
T0056 BOOL  ; NG拨料气缸缩回位延时
T0057 BOOL  ; NG拨料气缸伸出位延时
T0058 BOOL  ; 上料提升气缸缩回位延时
T0059 BOOL  ; 上料提升气缸伸出位延时
T0060 BOOL  ; 扫码NG缓存气缸缩回位延时
T0061 BOOL  ; 扫码NG缓存气缸伸出位延时
T0062 BOOL  ; 前机械手回#1腔体取料位延时
T0063 BOOL  ; 前机械手回#2腔体放料延时
T0064 BOOL  ; 前机械手回#2腔体取料延时
T0065 BOOL  ; 前机械手回#1腔体取料延时
T0066 BOOL  ; 前机械手回#2腔体取料延时
T0067 BOOL  ; 前机械手回OK位放料位延时
T0068 BOOL  ; 前机械手回左NG位延时
T0069 BOOL  ; 前机械手回右NG位延时
T0070 BOOL  ; 备用
T0071 BOOL  ; 备用
T0072 BOOL  ; 上料提升伸出位异常检测延时
T0073 BOOL  ; 上料提升伸出位异常检测延上料缩回延时检测
T0074 BOOL  ; 上左夹子闭合延时
T0075 BOOL  ; 上左夹张开报警延时
T0076 BOOL  ; 上右夹延时
T0077 BOOL  ; 上右夹张开延时
T0078 BOOL  ; 1合模伸出延时报警
T0079 BOOL  ; 1合模缩回延时报警
T0080 BOOL  ; 2合模伸出延时报警
T0081 BOOL  ; 2合模缩回延时报警
T0082 BOOL  ; 上料升降下降延时
T0083 BOOL  ; 上料升降回位延时
T0084 BOOL  ; 下料提升伸出位异常检测延时
T0085 BOOL  ; 下料提升缩回位异常检测延
T0086 BOOL  ; 右升降缸到位延时
T0087 BOOL  ; 右升降缸到位延时
T0088 BOOL  ; 下左夹闭合延时检测
T0089 BOOL  ; 下左夹张开延时检测
T0090 BOOL  ; 下右夹闭合报警延时
T0091 BOOL  ; 下右夹张开报警延时
T0092 BOOL  ; NG缩回异常延时
T0093 BOOL  ; NG伸出异常延时
T0094 BOOL  ; 私服ON报警延时
T0095 BOOL  ; 下料伺服异常延时
T0096 BOOL  ; 气压异常延时
T0097 BOOL  ; 电池流出出料拉带延时
T0098 BOOL  ; 右爪数据接收异常
T0099 BOOL  ; 左爪数据接收异常
T0100 BOOL  ; 扫码NG缸延时原位
T0101 BOOL  ; 扫码NG缸延时到位
T0102 BOOL  ; 下料位有料辅助
T0103 BOOL  ; NG下料位有料辅助
T0105 BOOL  ; 过度拉带末端有料持续信号
T0106 BOOL  ; 过渡拉带到移栽距离运动延时
T0107 BOOL  ; 上料无料感应延时
T0125 BOOL  ; 单料模式切换判断延时#1
T0126 BOOL  ; 单料模式切换判断延时#2
T0127 BOOL  ; 前右NG位按下时间
T0128 BOOL  ; 扫码气缸缩回报警
T0129 BOOL  ; 扫码气缸伸出报警
T0130 BOOL  ; #1复位破真空延时
T0131 BOOL  ; #1达到破真空持续时间
T0132 BOOL  ; #2复位破真空延时
T0133 BOOL  ; #2达到破真空持续时间
T0134 BOOL  ; #3复位破真空延时
T0135 BOOL  ; #3达到破真空持续时间
T0136 BOOL  ; #4复位破真空延时
T0137 BOOL  ; #4达到破真空持续时间
T0140 BOOL  ; 上料机械手Alarm_Clr输出时间
T0141 BOOL  ; 下料机械手Alarm_Clr输出时间
T0142 BOOL  ; 开机按钮持续时间
T0150 BOOL  ; 真空泵打开延时
T0151 BOOL  ; 真空泵断开延时
T0152 BOOL  ; #1腔体抽气时间
T0153 BOOL  ; #1腔体自检保压前延时
T0154 BOOL  ; #1腔体自检保压延时
T0155 BOOL  ; #2腔体抽气时间
T0156 BOOL  ; #2腔体自检保压前延时
T0157 BOOL  ; #2腔体自检保压延时
T0158 BOOL  ; 破真空阀打开延时
T0159 BOOL  ; 破真空阀打开延时
T0160 BOOL  ; 进料旋转回#1待料角度延时
T0161 BOOL  ; 进料旋转回#2待料位置延时
T0162 BOOL  ; 进料旋转回进料角度延时
T0163 BOOL  ; 出料旋转回#1待料角度延时
T0164 BOOL  ; 出料旋转回#2待料角度延时
T0165 BOOL  ; 出料旋转回下料角度延时
T0166 BOOL  ; 上料机械手到右爪上料位置延时
T0167 BOOL  ; 上料机械手回#1腔体位置
T0168 BOOL  ; 上料机械手回#2腔体位置
T0169 BOOL  ; 下料机械手回OK位置延时
T0170 BOOL  ; 下料机械手回NG位置延时
T0171 BOOL  ; 下料机械手回#1腔体位置延时
T0172 BOOL  ; 下料机械手回#2腔体位置延时
T0173 BOOL  ; 下料机械手回#4腔体放料延时
T0174 BOOL  ; 下料机械手回#4腔体取料延时
T0175 BOOL  ; 下料机械手回#3腔体取料延时
T0176 BOOL  ; 下料机械手回#4腔体取料延时
T0177 BOOL  ; 下料机械手回OK位放料位延时
T0178 BOOL  ; 下料机械手回左NG位延时
T0179 BOOL  ; 下料机械手回右NG位延时
T0180 BOOL  ; #1扫码后判断延时
T0181 BOOL  ; #2扫码后延时
T0183 BOOL  ; 上料轴到左上料位延时
T0184 BOOL  ; 下料轴回右OK下料位
T0190 BOOL  ; 氦检仪状体判断延时
T0191 BOOL  ; 检漏口压力判断延时
T0192 BOOL  ; 漏率判断延时
T0193 BOOL  ; 单元4串口1占用时间
T0200 BOOL  ; #1腔体抽气时间
T0201 BOOL  ; #1氦检阀打开延时
T0202 BOOL  ; 氦检持续时间
T0203 BOOL  ; #1延时
T0204 BOOL  ; 测试结束后抽残气延时
T0205 BOOL  ; 抽残气时间
T0206 BOOL  ; #1延时
T0207 BOOL  ; #1氦检阀打开抽气阀关闭延时
T0208 BOOL  ; 延时触发
T0209 BOOL  ; 扫码NG左槽
T0210 BOOL  ; #2腔体抽气时间
T0211 BOOL  ; #2氦检阀打开延时
T0212 BOOL  ; 氦检持续时间
T0213 BOOL  ; #2腔体数据传输延时
T0214 BOOL  ; 测试结束后抽残气延时
T0215 BOOL  ; 抽残气时间
T0216 BOOL  ; #2延时
T0217 BOOL  ; #2氦检阀打开抽气阀关闭延时
T0220 BOOL  ; 拉带有料持续时间
T0221 BOOL  ; 拉带无料持续时间
T0222 BOOL  ; 松爪后延时
T0230 BOOL  ; #1腔体复位破真空延时
T0231 BOOL  ; #1腔体达到破真空持续时间
T0232 BOOL  ; #2腔体复位破真空延时
T0233 BOOL  ; #2腔体达到破真空持续时间
T0240 BOOL  ; 拉带可放料信号延时
T0300 BOOL  ; 上料轴回左上料位
T0301 BOOL  ; 下料轴回右爪放OK位延时
T0306 BOOL  ; 上料机械手回进料位置延时
T0307 BOOL  ; 上料机械手回#1腔体位置延时
T0308 BOOL  ; 上料机械手回#2腔体位置延时
T0309 BOOL  ; 出料机械手回#1腔体位置延时
T0310 BOOL  ; 出料机械手回#2腔体位置延时
T0311 BOOL  ; 下料机械手回左爪OK位置延时
T0312 BOOL  ; 下料机械手回NG位置延时
T0313 BOOL  ; 进料旋转回进料反角度延时
T0314 BOOL  ; 后机械手右抓料气缸张开位时间
T0315 BOOL  ; 后机械手右抓料气缸夹紧位时间
T0316 BOOL  ; 后机械手升降气缸缩回位时间
T0317 BOOL  ; 后机械手升降气缸伸出位时间
T0318 BOOL  ; 后机械手左夹爪升降气缸缩回位时间
T0319 BOOL  ; 后机械手左夹爪升降气缸伸出位时间
T0320 BOOL  ; 氦检仪通信异常时间
T0321 BOOL  ; 1#扫码通信异常
T0322 BOOL  ; #1真空计断线延时
T0323 BOOL  ; #2真空计断线延时
T0324 BOOL  ; 上料机械手报警信号持续时间
T0325 BOOL  ; 下料机械手报警信号持续时间
T0326 BOOL  ; #3腔体移位气缸缩回位时间
T0327 BOOL  ; #3腔体移位气缸伸出位时间
T0328 BOOL  ; #4腔体移位气缸缩回位时间
T0329 BOOL  ; #4腔体移位气缸伸出位时间
T0330 BOOL  ; #1腔体顶升气缸缩回位时间
T0331 BOOL  ; #1腔体顶升气缸伸出位时间
T0332 BOOL  ; #2腔体顶升气缸缩回位时间
T0333 BOOL  ; #2腔体顶升气缸伸出位时间
T0334 BOOL  ; #3腔体顶升气缸缩回位时间
T0335 BOOL  ; #3腔体顶升气缸伸出位时间
T0336 BOOL  ; #4腔体顶升气缸缩回位时间
T0337 BOOL  ; #4腔体顶升气缸伸出位时间
T0338 BOOL  ; 前NG拨料气缸缩回位时间
T0339 BOOL  ; 前NG拨料气缸伸出位时间
T0340 BOOL  ; 后NG拨料气缸缩回位时间
T0341 BOOL  ; 后NG拨料气缸伸出位时间
T0342 BOOL  ; 进料舱门气缸缩回位时间
T0343 BOOL  ; 进料舱门气缸伸出位时间
T0344 BOOL  ; 出料舱门气缸缩回位时间
T0345 BOOL  ; 出料舱门气缸伸出位时间
T0350 BOOL  ; 系统运行延时
T0351 BOOL  ; 2#扫码通信异常
T0358 BOOL  ; NG槽满料感应延时
T0370 BOOL  ; 氦检仪不在检漏状态延时
T0400 BOOL  ; PC运行标志断开时间
T0401 BOOL  ; PC通信正常持续时间
T0402 BOOL  ; 前机械手左夹爪张开超时
T0403 BOOL  ; 前机械手左夹爪夹紧超时
T0404 BOOL  ; 前机械手右夹爪张开超时
T0405 BOOL  ; 前机械手右夹爪夹紧超时
T0406 BOOL  ; 前机械手升降气缸缩回超时
T0407 BOOL  ; 前机械手升降气缸伸出超时
T0408 BOOL  ; 前机械手左夹爪升降气缸缩回超时
T0409 BOOL  ; 前机械手左夹爪升降气缸伸出超时
T0410 BOOL  ; 前机械手右夹爪升降气缸缩回超时
T0411 BOOL  ; 前机械手右夹爪升降气缸伸出超时
T0412 BOOL  ; 后机械手左抓料气缸张开超时
T0413 BOOL  ; 后机械手左抓料气缸夹紧超时
T0414 BOOL  ; 后机械手右抓料气缸张开超时
T0415 BOOL  ; 后机械手右抓料气缸夹紧超时
T0416 BOOL  ; 后机械手升降气缸缩回超时
T0417 BOOL  ; 后机械手升降气缸伸出超时
T0418 BOOL  ; 后机械手左夹爪升降气缸缩回超时
T0419 BOOL  ; 后机械手左夹爪升降气缸伸出超时
T0420 BOOL  ; 后机械手右夹爪升降气缸缩回超时
T0421 BOOL  ; 后机械手右夹爪升降气缸伸出超时
T0422 BOOL  ; #1腔体移位气缸缩回超时
T0423 BOOL  ; #1腔体移位气缸伸出超时
T0424 BOOL  ; #2腔体移位气缸缩回超时
T0425 BOOL  ; #2腔体移位气缸伸出超时
T0426 BOOL  ; #3腔体移位气缸缩回超时
T0427 BOOL  ; #3腔体移位气缸伸出超时
T0428 BOOL  ; #4腔体移位气缸缩回超时
T0429 BOOL  ; #4腔体移位气缸伸出超时
T0430 BOOL  ; #1腔体顶升气缸缩回超时
T0431 BOOL  ; #1腔体顶升气缸伸出超时
T0432 BOOL  ; #2腔体顶升气缸缩回超时
T0433 BOOL  ; #2腔体顶升气缸伸出超时
T0434 BOOL  ; #3腔体顶升气缸缩回超时
T0435 BOOL  ; #3腔体顶升气缸伸出超时
T0436 BOOL  ; #4腔体顶升气缸缩回超时
T0437 BOOL  ; #4腔体顶升气缸伸出超时
T0438 BOOL  ; 前NG拨料气缸缩回超时
T0439 BOOL  ; 前NG拨料气缸伸出 超时
T0440 BOOL  ; 后NG拨料气缸缩回超时
T0441 BOOL  ; 后NG拨料气缸伸出超时
T0442 BOOL  ; 进料舱门气缸缩回超时
T0443 BOOL  ; 进料舱门气缸伸出超时
T0444 BOOL  ; 出料舱门气缸缩回超时
T0445 BOOL  ; 出料舱门气缸伸出超时
T0450 BOOL  ; 氦检仪漏率低于设定值延时
T0451 BOOL  ; 氦检漏率正常判断时间
T0456 BOOL  ; 延时关校准
T0500 BOOL  ; 上料横移气缸异常信息持续时间
T0501 BOOL  ; 上料横移气缸伸出异常信息持续时间
T0502 BOOL  ; 上料旋转位异常信心持续时间
T0503 BOOL  ; 上料提升气缸不在原位信息持续时间
T0504 BOOL  ; 上料移栽气缸不在伸出位信息持续时间
T0505 BOOL  ; 上料提升气缸不在伸出位信息持续时间
T0506 BOOL  ; 上料升降气缸不在伸出位信息持续时间
T0507 BOOL  ; 进料移栽气缸动作异常信息持续时间
T0508 BOOL  ; 进料旋转归零异常信息持续时间
T0509 BOOL  ; 上料升降气缸不在原位异常信息持续时间
T0510 BOOL  ; 上料旋转没归零异常
T0511 BOOL  ; 进料移栽缩回异常信息持续时间
T0512 BOOL  ; 上料移栽没伸出信息持续时间
T0513 BOOL  ; 进料提升气缸没缩回信息持续时间
T0520 BOOL  ; 下料提升气缸不在原位信息持续时间
T0521 BOOL  ; 下料升降气缸不在原位信息持续时间
T0522 BOOL  ; 下料横移气缸不在伸出位信息持续时间
T0524 BOOL  ; 下料提升气缸不在原位信息持续时间
T0525 BOOL  ; 下料移栽气缸不在伸出位信息持续时间
T0526 BOOL  ; 上料提升气缸不在伸出位信息持续时间
T0527 BOOL  ; 升降气缸不在伸出位信息持续时间
T0528 BOOL  ; 下料移栽气缸动作异常信息持续时间
T0529 BOOL  ; 下料旋转运动异常信息持续时间
T0530 BOOL  ; 下料升降气缸不在原位异常信息持续时间
T0531 BOOL  ; 下料旋转没归零异常
T0540 BOOL  ; 进料提升气缸不在原位信息持续时间
T0541 BOOL  ; 出料提升气缸不在原位信息持续时间
T0542 BOOL  ; #1腔体真空值大于破真空设定值信息持续事假
T0543 BOOL  ; #1抽气阀打开异常信息持续时间
T0544 BOOL  ; #1氦检阀打开异常信息持续时间
T0545 BOOL  ; #1破真空阀打开异常信息持续时间
T0546 BOOL  ; #1吹气阀打开异常信息持续时间
T0547 BOOL  ; 进料提升气缸不在原位异常信息持续时间
T0548 BOOL  ; 出料提升气缸不在原位异常信息持续时间
T0549 BOOL  ; #2腔体真空值大于破真空设定值信息持续时间
T0550 BOOL  ; #2抽气阀异常信息持续时间
T0551 BOOL  ; #2氦检阀异常信息持续时间
T0552 BOOL  ; #2破真空阀异常信息持续时间
T0553 BOOL  ; #2吹气阀异常信息持续时间
T0560 BOOL  ; 进料机械手位置异常信息持续时间
T0561 BOOL  ; 上料旋转位置异常信息持续时间
T0562 BOOL  ; 进料夹爪松开异常信息持续时间
T0563 BOOL  ; #1合模气缸不在缩回位异常信息持续时间
T0564 BOOL  ; 进料夹爪不在张开位异常信息持续时间
T0565 BOOL  ; #2合模气缸不在缩回位异常信息持续时间
T0566 BOOL  ; 进料夹爪不在张开位异常信息持续时间
T0567 BOOL  ; 进料提升气缸不在伸出位异常信息持续时间
T0568 BOOL  ; 进料提升气缸不在缩回位异常信息持续时间
T0569 BOOL  ; 进料机械手没归零异常信息持续时间
T0570 BOOL  ; 进料机械手到达左极限信息持续时间
T0571 BOOL  ; 进料机械手到达右极限信息持续时间
T0572 BOOL  ; 出料机械手避让位置异常信息持续时间
T0573 BOOL  ; 出料机械手避让位置异常信息持续时间
T0580 BOOL  ; 出料机械手位置异常信息持续时间
T0581 BOOL  ; 下料旋转气缸位置异常信息持续时间
T0582 BOOL  ; 下料缓存有料异常信息持续时间
T0583 BOOL  ; #1合模气缸不在缩回位异常信息持续时间
T0584 BOOL  ; #2合模气缸不在缩回位异常信息持续时间
T0585 BOOL  ; 出料夹爪不在张开位异常信息持续时间
T0586 BOOL  ; 出料提升气缸不在伸出位异常信息持续时间
T0587 BOOL  ; 出料提升气缸不在缩回位异常信息持续时间
T0588 BOOL  ; 出料机械手没归零异常信息持续时间
T0589 BOOL  ; 出料机械手到达左极限异常信息持续时间
T0590 BOOL  ; 出料机械手到达右极限异常信息持续时间
T0591 BOOL  ; 进料机械手位置避让异常信息持续时间
T0592 BOOL  ; 进料机械手位置避让异常信息持续时间
T0600 BOOL  ; 出料旋转位无料延时
T0610 BOOL  ; 扫码气缸原位延时
T0611 BOOL  ; 扫码气缸到位延时
T0622 BOOL  ; 氦捡仪稳定时间
T0627 BOOL  ; 空气进化器延时关闭
T0631 BOOL  ; #1抽气阀打开延时(A)
T0633 BOOL  ; #2抽气阀打开延时(A)
T0640 BOOL  ; #1腔体破真空值到达
T0641 BOOL  ; #1腔氦检阀关闭延时
T0650 BOOL  ; #2腔体破真空值到达
T0651 BOOL  ; #2腔氦检阀关闭延时
T0700 BOOL  ; 腔体无料信号
T0755 BOOL  ; 抽残气打开延时
T0756 BOOL  ; #2抽残气打开延时
T0770 BOOL  ; 延时触发
T0771 BOOL  ; 延时触发2
T0772 BOOL  ; 延时触发3
T0773 BOOL  ; 下料安全为没料感应延时
T0774 BOOL  ; 清料
T0775 BOOL  ; 电脑未启动/屏蔽
T0776 BOOL  ; 电脑未启动/屏蔽
T0777 BOOL  ; 电脑未启动/屏蔽
T0780 BOOL  ; 电脑未启动/屏蔽
T0781 BOOL  ; 电脑未启动/屏蔽
T0782 BOOL  ; 校验通信异常
T0791 BOOL  ; 上料位异常延时
T0792 BOOL  ; 清掉上料位有料时间
T0794 BOOL  ; 拉带暂停时扫码延时
T0796 BOOL  ; 重复扫码时间
T0799 BOOL  ; 柔性复位
T0800 BOOL  ; 复位按钮2秒延时
T0801 BOOL  ; 复位完提示
T0802 BOOL  ; 扫码位有料信号
T0803 BOOL  ; 扫码位料停留延时
T0804 BOOL  ; s扫码位料流走检测
T0805 BOOL  ; 上料位待料延时
T0806 BOOL  ; 延时辅助1
T0807 BOOL  ; 下料延时辅助2
T0809 BOOL  ; 回位辅助
T0810 BOOL  ; 右下料数据交互延时判断
T0811 BOOL  ; 左传输超时
T0812 BOOL  ; 带料触发复位
T0813 BOOL  ; 到腔体判断时间
T0814 BOOL  ; 下料延时
T0820 BOOL  ; 接触器动作时间
T0821 BOOL  ; 按键时间
T0822 BOOL  ; 扫码不良料取走延时
T0823 BOOL  ; 吹气破真空延时
T0824 BOOL  ; 扫码位—上料位料流动延时检测
T0825 BOOL  ; 下一步
T0826 BOOL  ; 下一步
T0827 BOOL  ; 延时辅助
T0828 BOOL  ; FZ2
T0829 BOOL  ; 破真空时真空计2异常检测延时
T0830 BOOL  ; 报警音
T0831 BOOL  ; 真空计破真空异常辅助
T0833 BOOL  ; 强制清料
T0851 BOOL  ; 氦检阀1关闭检测延时
T0852 BOOL  ; 氦检阀2关闭检测延时
T0853 BOOL  ; 下料区电池流出安全区延时
T0900 BOOL  ; ts
T0901 BOOL  ; ts1
T0912 BOOL  ; 清料时间
T1000 BOOL  ; 上料位有料
T1258 BOOL  ; 破真空阀打开延时
W0.00 BOOL  ; 手/自动切换HMI
W0.01 BOOL  ; 开机初始状态
W0.14 BOOL  ; 复位按钮-HMI
W0.15 BOOL  ; 清料停机-HMI
W100.00 BOOL  ; 气缸下降安全位置
W100.01 BOOL  ; 下料气缸安全位置
W100.02 BOOL  ; 上料轴2级气缸安全位置
W100.03 BOOL  ; 下料升降安全位置
W100.05 BOOL  ; s
W101.00 BOOL  ; 记忆有料标志
W101.01 BOOL  ; 手动记忆有料启动异常
W102.00 BOOL  ; 右爪抓料
W102.01 BOOL  ; 左爪抓料
W10.00 BOOL  ; 上料机械手回NG槽安全条件
W10.01 BOOL  ; 放料位安全条件
W10.03 BOOL  ; 单料模式下判断夹爪下料位置辅助
W110.00 BOOL  ; 程序强制清除
W119.15 BOOL  ; 氦捡仪稳定中
W12.02 BOOL  ; #1合模气缸手动缩回
W12.08 BOOL  ; #2合模气缸手动缩回
W12.13 BOOL  ; #1腔体自检条件
W12.14 BOOL  ; #1腔体自检中
W12.15 BOOL  ; #1合模气缸自检伸出
W13.00 BOOL  ; #1抽气阀自检输出
W13.01 BOOL  ; #1腔体自检进入保压前状态
W13.02 BOOL  ; #1腔体自检进入保压状态
W13.03 BOOL  ; #1腔体保压结束
W13.05 BOOL  ; #1腔体自检破真空阀打开
W13.07 BOOL  ; #1腔体自检破真空结束
W13.08 BOOL  ; #1腔体自检吹气阀打开
W13.09 BOOL  ; #1腔体自检结束
W13.10 BOOL  ; #2腔体自检条件
W13.11 BOOL  ; #2腔体自检中
W13.12 BOOL  ; #2合模气缸自检伸出
W13.13 BOOL  ; #2抽气阀自检输出
W13.14 BOOL  ; #2腔体自检进入保压前状体
W13.15 BOOL  ; #2腔体自检进入保压状态
W14.00 BOOL  ; #2腔体保压结束
W14.01 BOOL  ; #2腔体自检破真空阀打开
W14.02 BOOL  ; #2腔体自检破真空结束
W14.03 BOOL  ; #2腔体自检吹气阀打开
W14.04 BOOL  ; #2腔体自检结束
W14.05 BOOL  ; #2合模气缸缩回
W14.06 BOOL  ; #1合模气缸缩回
W14.10 BOOL  ; 氦检仪不在检漏状态
W14.15 BOOL  ; 氦捡仪稳定中
W150.00 BOOL  ; 校准完成
W150.01 BOOL  ; 校准出错
W15.00 BOOL  ; 上料扫码左NG槽手动
W15.01 BOOL  ; 上料扫码右NG槽手动
W15.02 BOOL  ; 校准中
W15.05 BOOL  ; 上料手动到左爪上料位置
W15.06 BOOL  ; 上料机械手手动归零
W15.07 BOOL  ; 上料机械手手动左移
W15.08 BOOL  ; 上料机械手手动右移
W15.09 BOOL  ; 进料机械手手动到右爪上料位置
W15.10 BOOL  ; 上料机械手手动到腔体1位置
W15.11 BOOL  ; 上料机械手手动到腔体2位置
W16.00 BOOL  ; 下料提升气缸伸出条件
W16.01 BOOL  ; 下料提升气缸手动伸出
W16.04 BOOL  ; 下料轴回右爪下OK位置
W16.05 BOOL  ; 出料轴手动到右OK位置
W16.06 BOOL  ; 下料机械手手动归零
W16.07 BOOL  ; 下料机械手手动左移
W16.08 BOOL  ; 下料机械手手动右移
W16.09 BOOL  ; 出料轴手动到左OK位置
W16.10 BOOL  ; 下料机械手手动到NG下料位
W16.11 BOOL  ; 下料机械手手动到腔体1位置
W16.12 BOOL  ; 下料机械手手动到腔体2位置
W17.06 BOOL  ; 上料机械手回右爪上料位置
W17.07 BOOL  ; 上料机械手回#1腔体位置
W17.08 BOOL  ; 上料机械手回#2腔体位置
W17.09 BOOL  ; 下料机械手回左爪OK位置
W17.10 BOOL  ; 下料机械手回NG位置
W17.11 BOOL  ; 下料机械手回#1腔体位置
W17.12 BOOL  ; 下料机械手回#2腔体位置
W19.10 BOOL  ; 启动状态
W19.15 BOOL  ; 氦检仪启动
W1.00 BOOL  ; 扫码阻挡—HMI 伸出
W1.01 BOOL  ; 扫码阻挡缩回HMI
W1.02 BOOL  ; 进料输送电机HMI
W1.03 BOOL  ; NG气缸HMI
W1.04 BOOL  ; 出料输送电机HMI
W1.05 BOOL  ; 扫码阻挡（HMI）
W1.09 BOOL  ; 扫码NG缸 HMI
W200.00 BOOL  ; 调试
W200.06 BOOL  ; TS
W20.00 BOOL  ; #1电池扫码信号
W21.09 BOOL  ; 进料旋转回#1待料角度
W21.10 BOOL  ; 进料旋转回#2待料角度
W21.11 BOOL  ; 进料旋转回进料角度
W21.14 BOOL  ; 进料旋转回进料反角度
W22.00 BOOL  ; 上料轴自动去左爪上料位
W22.03 BOOL  ; 上料机械手到#1腔体
W22.04 BOOL  ; 上料机械手到#2腔体
W22.08 BOOL  ; 上料轴从腔体1回右爪上料位置
W22.09 BOOL  ; 上料机械手归零后回上料位置
W22.10 BOOL  ; 上料轴从腔体2回右上料位
W22.13 BOOL  ; 到扫码NG槽（右） 下料轴到NG槽
W22.14 BOOL  ; 到扫码NG槽（左） 下料轴到NG槽
W23.00 BOOL  ; 合模气缸1伸出
W23.01 BOOL  ; #1抽气阀打开
W23.02 BOOL  ; #1抽气结束
W23.03 BOOL  ; #1氦检阀打开
W23.04 BOOL  ; #1氦检正常结束
W23.05 BOOL  ; #1抽气异常结束
W23.06 BOOL  ; #1抽气阀关闭
W23.07 BOOL  ; #1抽气阀打开(抽残气)
W23.08 BOOL  ; #1抽残气结束
W23.09 BOOL  ; #1腔体破真空阀打开
W23.10 BOOL  ; #1腔体破真空结束
W23.11 BOOL  ; #1腔体吹气阀打开
W23.12 BOOL  ; #1合模气缸缩回
W23.13 BOOL  ; 腔体1关闭条件
W23.14 BOOL  ; 氦检异常
W24.00 BOOL  ; 合模气缸2伸出
W24.01 BOOL  ; #2抽气阀打开
W24.02 BOOL  ; #2抽气结束
W24.03 BOOL  ; #2氦检阀打开
W24.04 BOOL  ; #2氦检正常结束
W24.05 BOOL  ; #2抽气异常结束
W24.06 BOOL  ; #2抽气阀关闭
W24.07 BOOL  ; #2抽气阀打开(抽残气)
W24.08 BOOL  ; #2抽残气结束
W24.09 BOOL  ; #2腔体破真空阀打开
W24.10 BOOL  ; #2腔体破真空结束
W24.11 BOOL  ; #2腔体吹气阀打开
W24.12 BOOL  ; #2合模气缸缩回
W24.13 BOOL  ; 合模气缸2伸出条件
W24.14 BOOL  ; #2氦检异常
W25.00 BOOL  ; 下料机械手回#1腔体位置
W25.01 BOOL  ; 下料机械手回#2腔体位置
W25.05 BOOL  ; 下料轴回右爪OK位置
W25.06 BOOL  ; 下料机械手回左爪OK位置
W25.07 BOOL  ; 下料机械手回NG位置辅助1
W25.08 BOOL  ; 下料机械手回NG位置辅助2
W25.13 BOOL  ; 下料机械手归零后回左OK位
W26.00 BOOL  ; 出料旋转回#1出料位
W26.13 BOOL  ; 出料旋转回#2出料角度
W26.14 BOOL  ; 出料旋转回出料角度
W27.00 BOOL  ; 出料旋转归零后回下料角度
W28.00 BOOL  ; 上料轴回左爪上料位置
W28.01 BOOL  ; 下料轴自动回右爪ok位置
W28.02 BOOL  ; 下料轴自动回左爪放料位
W28.06 BOOL  ; 上料机械手回右爪进料位置
W28.07 BOOL  ; 上料机械手回#1腔体位置
W28.08 BOOL  ; 上料机械手回#2腔体位置
W28.09 BOOL  ; 下料机械手回#1腔体位置
W28.10 BOOL  ; 下料机械手回#2腔体位置
W28.11 BOOL  ; 下料机械手回左爪OK位置
W28.12 BOOL  ; 下料机械手回NG位置
W2.01 BOOL  ; 下料提升HMI
W2.02 BOOL  ; 下料升降HMI
W2.03 BOOL  ; 下料左夹爪HMI
W2.04 BOOL  ; 下料右夹爪HMI
W300.00 BOOL  ; 设备故障
W303.01 BOOL  ; 设备暂停
W30.00 BOOL  ; #1电池扫码完成
W30.01 BOOL  ; #1扫码失败
W30.02 BOOL  ; #1扫码OK
W30.04 BOOL  ; 取料位电池扫码NG
W30.05 BOOL  ; 取料位电池扫码OK
W30.06 BOOL  ; 手动输入条码
W30.10 BOOL  ; 校验OK
W30.11 BOOL  ; 校验NG
W310 CHANNEL  ; 复位w310后设置位数
W310.00 BOOL  ; 扫码阻挡伸出辅助1
W310.01 BOOL  ; 上料提升辅助
W310.02 BOOL  ; 上料升降辅助（左）
W310.03 BOOL  ; 真空泵辅助1
W310.04 BOOL  ; 上料左夹爪辅助1
W310.05 BOOL  ; 上料右夹爪
W310.06 BOOL  ; #2上料升降辅助（右）
W310.07 BOOL  ; #2下料升降气缸辅助
W310.10 BOOL  ; 氦检1抽真空辅助1
W310.11 BOOL  ; 氦检1氦检阀辅助1
W310.12 BOOL  ; 氦检1破真空辅助1
W310.13 BOOL  ; 氦检1吹气辅助1
W310.14 BOOL  ; 氦检2抽真空阀辅助1
W310.15 BOOL  ; 氦检2氦检阀辅助1
W311 CHANNEL  ; 复位311指定起始位及位数
W311.00 BOOL  ; 氦检2破真空辅助
W311.01 BOOL  ; 氦检2吹气辅助
W311.02 BOOL  ; 上料阻挡
W311.03 BOOL  ; 扫码阻挡伸出辅助
W311.04 BOOL  ; 下料提升气缸辅助1
W311.05 BOOL  ; 扫码阻挡
W311.06 BOOL  ; 下料左夹爪辅助1
W311.07 BOOL  ; 下料右夹爪辅助1
W311.08 BOOL  ; NG气缸辅助1
W311.09 BOOL  ; 进料输送电机
W311.10 BOOL  ; 出料输送带辅助1
W311.11 BOOL  ; 出料输送带辅助2
W311.12 BOOL  ; 手动操作限制
W311.13 BOOL  ; 操作限制2
W311.14 BOOL  ; 下料轴动作
W311.15 BOOL  ; 备用
W312.00 BOOL  ; 启动指示灯辅助
W312.01 BOOL  ; 停止指示灯辅助1
W312.02 BOOL  ; 复位指示灯
W312.03 BOOL  ; 三色灯红辅助1
W312.04 BOOL  ; 三色灯绿辅助1
W312.05 BOOL  ; 三色黄灯辅助1
W312.06 BOOL  ; 蜂鸣器辅助1
W312.07 BOOL  ; 蜂鸣器辅助2
W312.08 BOOL  ; 扫码NG气缸辅助1
W312.10 BOOL  ; 扫码NG缸辅助
W313.00 BOOL  ; 氦检仪启动辅助1
W314.00 BOOL  ; 手动操作限制3
W314.01 BOOL  ; 手动操作限制4
W315.09 BOOL  ; 备用
W328.00 BOOL  ; 扫码阻挡气缸辅助（手动）
W329.00 BOOL  ; 上料私服使能
W329.01 BOOL  ; 下料伺服使能辅助1
W32.00 BOOL  ; 读检漏仪状态
W32.01 BOOL  ; 读氦检仪状态完成
W32.02 BOOL  ; 读检漏口压力
W32.03 BOOL  ; 读检漏口压力完成
W32.05 BOOL  ; 读漏率
W32.06 BOOL  ; 读漏率完成
W32.07 BOOL  ; 读漏率失败
W32.08 BOOL  ; 读氦检仪状态失败
W32.09 BOOL  ; 读检漏口压力失败
W332.00 BOOL  ; 氦检仪电源启动辅助
W339.00 BOOL  ; 备用5
W34.00 BOOL  ; 氦检仪当前为检漏状态
W34.01 BOOL  ; 氦检仪当前为待机状态
W34.02 BOOL  ; 氦检仪当前为启动状态
W34.03 BOOL  ; 氦检仪当前为定标状态
W34.04 BOOL  ; 氦检仪当前为错误状态
W34.05 BOOL  ; 氦检仪当前为暂停状态
W34.15 BOOL  ; 氦捡仪稳定中
W380.00 BOOL  ; 强制清除有料记忆
W380.02 BOOL  ; 上料模式选择HMI（1或2）
W390.00 BOOL  ; 暂停 继续
W390.01 BOOL  ; 安全门信号
W390.02 BOOL  ; 拉带2手自动切换按钮HMI
W390.03 BOOL  ; 拉带2手自动
W395.00 BOOL  ; 真空泵异常
W399.00 BOOL  ; 单料模式
W399.09 BOOL  ; 总复位HMI
W39.00 BOOL  ; 上料机械手在原点位
W39.01 BOOL  ; 下料机械手在原点位
W3.00 BOOL  ; 机械手归零-HMI
W3.01 BOOL  ; 上料机械手左移按钮-HMI
W3.02 BOOL  ; 上料机械手机械手右移按钮-HMI
W3.03 BOOL  ; 右爪上料位置-HMI
W3.04 BOOL  ; 腔体1位置-HMI
W3.05 BOOL  ; 腔体2位置-HMI
W3.06 BOOL  ; 进料提升气缸-HMI
W3.07 BOOL  ; 上左夹爪-HMI
W3.08 BOOL  ; 上右夹爪-HMI
W3.09 BOOL  ; #3上料夹爪-HMI
W3.10 BOOL  ; #4上料夹爪-HMI
W3.11 BOOL  ; 上料升降HMI
W3.12 BOOL  ; 左爪上料位置-HMI
W3.13 BOOL  ; 右爪上料位置
W3.14 BOOL  ; 右上料升降HMI
W400 CHANNEL  ; 复位W400.00-W409.15
W400.00 BOOL  ; 总复位信号
W400.01 BOOL  ; 复位中
W400.02 BOOL  ; 复位完成
W400.03 BOOL  ; 自动中
W400.04 BOOL  ; 不允许往下放料标志
W400.05 BOOL  ; 停机
W400.06 BOOL  ; 第一个料
W400.07 BOOL  ; 输送带自动中
W400.08 BOOL  ; 扫码位料先到
W400.09 BOOL  ; 扫码OK料已流走
W400.10 BOOL  ; 运行时程序第复位结束标志
W400.15 BOOL  ; 长输送带自动中
W401.00 BOOL  ; 有料信号有料不能复位弹窗
W401.01 BOOL  ; 腔体记忆有料不能复位
W401.02 BOOL  ; 爪子记忆有料不能复位
W401.03 BOOL  ; 腔体有料记忆不能复位
W401.05 BOOL  ; 扫码位有料记忆
W405.00 BOOL  ; 气缸复位步
W405.01 BOOL  ; 达复位
W405.02 BOOL  ; 腔体复位
W405.03 BOOL  ; 复位完成
W405.04 BOOL  ; 复位完成 退出
W405.05 BOOL  ; 上料马达回右爪上料步
W405.10 BOOL  ; 上料轴自动中
W405.11 BOOL  ; 下料轴自动中
W406.00 BOOL  ; 马达启动
W406.01 BOOL  ; 判断下一步动作
W406.02 BOOL  ; 往下放料
W406.03 BOOL  ; 退出传送循环送料
W406.05 BOOL  ; 左夹料位
W406.06 BOOL  ; 右夹爪有料取料步骤
W406.07 BOOL  ; 夹料步
W406.08 BOOL  ; 气缸上升
W406.09 BOOL  ; 去左爪取料位
W406.10 BOOL  ; 左爪去取料
W406.11 BOOL  ; 提升气缸缩回
W406.12 BOOL  ; 准备去放料
W406.13 BOOL  ; 上料放料判断步
W406.14 BOOL  ; 去1#腔体
W406.15 BOOL  ; 去2#腔体
W407.01 BOOL  ; 下料两个气缸同时下降
W407.02 BOOL  ; 开夹子
W407.03 BOOL  ; 气缸回缩
W407.04 BOOL  ; 回右夹爪取料位置
W407.05 BOOL  ; 设置两气缸下降
W407.06 BOOL  ; 2号腔体开夹子
W407.07 BOOL  ; 上升
W407.08 BOOL  ; 从2号腔体回右夹爪取料位置
W407.09 BOOL  ; 跳出上料自动循环
W407.10 BOOL  ; 空步
W407.11 BOOL  ; 扫码NG提升气缸下降
W407.12 BOOL  ; 提升缸上升
W407.13 BOOL  ; 推料步
W407.15 BOOL  ; 进入自动取料判断
W408.00 BOOL  ; 下料轴去腔体2取料
W408.01 BOOL  ; 下料升降气缸下降取料
W408.02 BOOL  ; 取料夹子夹料
W408.03 BOOL  ; 下料气缸提升
W408.04 BOOL  ; 测试结果传递 标志位设置
W408.05 BOOL  ; 下料位置判断
W408.06 BOOL  ; 放ok料步
W408.07 BOOL  ; 下料提升气缸下降
W408.08 BOOL  ; 气缸收回
W408.09 BOOL  ; 去左位放料
W408.10 BOOL  ; 判断可否下料
W408.11 BOOL  ; 开爪放料
W408.12 BOOL  ; 上升
W408.13 BOOL  ; T通讯判断
W408.14 BOOL  ; 退出自动步骤
W408.15 BOOL  ; 下料自动结束
W409.00 BOOL  ; 去腔体1取料
W409.01 BOOL  ; 取腔体1 气缸下降步
W409.02 BOOL  ; 取料夹子夹料
W409.03 BOOL  ; 腔体1取料 取料提升
W409.04 BOOL  ; 腔体1结果传递
W409.05 BOOL  ; 下料位置判断
W409.06 BOOL  ; 放NG料步
W409.07 BOOL  ; 放NG料
W409.08 BOOL  ; 放NG 下降 放料
W409.09 BOOL  ; 放NG 气缸上升
W409.10 BOOL  ; 推料步骤
W40.00 BOOL  ; 扫码右NG槽位
W40.01 BOOL  ; 扫码NG左槽
W40.02 BOOL  ; 回到初始位置
W40.03 BOOL  ; 左上料位
W410.00 BOOL  ; 拉带允许下料信号
W410.01 BOOL  ; 开始扫码
W410.02 BOOL  ; 扫码完成
W410.05 BOOL  ; 扫码II
W411.00 BOOL  ; 下料右爪数据更新请求
W411.01 BOOL  ; 右数据传送完成
W411.02 BOOL  ; 右爪下料通讯超时
W411.03 BOOL  ; 下料左爪数据传送请求
W411.04 BOOL  ; 左数据传送完成
W411.05 BOOL  ; 左爪下料通讯超时
W412.00 BOOL  ; 准备放右爪料
W412.01 BOOL  ; 左爪放料准备
W412.02 BOOL  ; NG料满 无法放NG料
W412.03 BOOL  ; 左放料延时等待
W412.04 BOOL  ; 料流走延时
W413.00 BOOL  ; 1#腔体自动开始
W413.01 BOOL  ; 抽真空
W413.02 BOOL  ; 氦检步骤
W413.03 BOOL  ; 清除NG料满 HMI
W413.04 BOOL  ; 关氦检 抽残气
W413.05 BOOL  ; 破真空
W413.06 BOOL  ; 停止吹气
W413.07 BOOL  ; 复位自动
W413.08 BOOL  ; 空步
W414.00 BOOL  ; 2#腔体自动开始
W414.01 BOOL  ; 抽真空
W414.02 BOOL  ; 氦检步骤
W414.04 BOOL  ; 关氦检 抽残气
W414.05 BOOL  ; 破真空
W414.06 BOOL  ; 停止吹气
W414.07 BOOL  ; 复位自动
W414.08 BOOL  ; 空步
W416.00 BOOL  ; 腔体1抽真空标志
W416.01 BOOL  ; 腔体2抽真空标志
W416.02 BOOL  ; 腔体1氦检中
W416.03 BOOL  ; 腔体2氦检中
W417.00 BOOL  ; 1真空计错误
W417.01 BOOL  ; 2真空计或破真空异常
W420.00 BOOL  ; 上料位有料
W420.01 BOOL  ; 左夹子上料柔性异常
W420.02 BOOL  ; 左夹子上料柔性异常报警辅助1
W420.03 BOOL  ; 1#放料柔性报警辅助
W420.04 BOOL  ; 放腔体1柔性异常
W420.05 BOOL  ; 2#放料柔性报警辅助
W420.06 BOOL  ; 放腔体2柔性异常
W420.07 BOOL  ; #2腔体取料柔性异常辅助
W420.08 BOOL  ; #2腔体放料柔性异常
W420.09 BOOL  ; 1#腔体取料柔性异常辅助
W420.10 BOOL  ; 1#腔体放料柔性异常
W420.11 BOOL  ; 右爪放ok料柔性异常辅助
W420.12 BOOL  ; 右爪放ok料柔性异常
W420.13 BOOL  ; 左爪放ok料柔性异常辅助
W420.14 BOOL  ; 左爪放ok料柔性异常
W420.15 BOOL  ; 放NG料柔性异常辅助
W421.01 BOOL  ; 放NG料柔性异常
W421.02 BOOL  ; 腔体1放料后有料感应异常
W421.03 BOOL  ; 腔体1取料后有料信号异常
W421.04 BOOL  ; 腔体1无料状态跟有料信号不一致
W421.05 BOOL  ; 腔体2无料状态跟有料信号不一致
W421.06 BOOL  ; 2#腔体放料后腔体有料信号异常
W421.07 BOOL  ; 2#腔体取料后腔体有料信号异常
W421.08 BOOL  ; 扫码位料流动到上料位异常
W421.09 BOOL  ; 右爪放OK料有料信号异常
W421.10 BOOL  ; 左爪放OK料有料感应异常
W421.11 BOOL  ; 1#爪取料后上料位有料状态跟有料信号不一致
W421.12 BOOL  ; 2#爪取料后上料位有料状态
W421.15 BOOL  ; 放扫码料柔性异常
W422.07 BOOL  ; 氦检仪检漏口 值长时超低
W430.00 BOOL  ; 扫码NG 下料位有料异常
W430.01 BOOL  ; NG 下料位有料异常
W430.03 BOOL  ; 扫码NG槽料满
W430.12 BOOL  ; 氦检阀1关闭异常
W430.13 BOOL  ; 氦检阀2关闭异常
W430.14 BOOL  ; 下料区电池流出超时
W430.15 BOOL  ; 下料区有料状态与信号不符
W44.00 BOOL  ; #1抽残气标志
W44.01 BOOL  ; #2抽残气
W44.02 BOOL  ; 计时辅助
W44.03 BOOL  ; #2计时辅助
W45.01 BOOL  ; 伺服复位
W48.00 BOOL  ; 启动辅助1
W48.01 BOOL  ; 启动辅助2
W48.02 BOOL  ; 启动辅助3
W48.03 BOOL  ; 启动辅助4
W48.04 BOOL  ; 启动辅助5
W48.05 BOOL  ; 启动条件满足
W49.00 BOOL  ; 报警清除HMI
W49.01 BOOL  ; NG报警清除HMI
W4.00 BOOL  ; 机械手归零-HMI
W4.01 BOOL  ; 下料机械手左移按钮-HMI
W4.02 BOOL  ; 下料机械手右移按钮-HMI
W4.03 BOOL  ; 下料轴左爪OK下料位置-HMI
W4.04 BOOL  ; NG下料位置-HMI
W4.05 BOOL  ; 腔体1位置-HMI
W4.06 BOOL  ; 腔体2位置-HMI
W4.07 BOOL  ; 下料提升气缸-HMI
W4.08 BOOL  ; 下左爪HMI
W4.09 BOOL  ; 下右爪HMI
W4.10 BOOL  ; #3出料夹爪-HMI
W4.11 BOOL  ; 下料升降HMI
W4.12 BOOL  ; 下料右爪OK下料位置-HMI
W4.13 BOOL  ; 下料轴右爪OK下料位—HMI
W500.00 BOOL  ; TS
W500.01 BOOL  ; ts2
W500.02 BOOL  ; ts3
W500.03 BOOL  ; ts3
W500.04 BOOL  ; ts5
W500.05 BOOL  ; ts5
W500.06 BOOL  ; TS6
W500.07 BOOL  ; ts7
W500.08 BOOL  ; TS
W500.09 BOOL  ; TS9
W500.10 BOOL  ; 调试
W500.11 BOOL  ; 调试
W500.15 BOOL  ; 清料
W501.00 BOOL  ; 强制开上料右夹子—HMI
W501.01 BOOL  ; 上左-HMI
W501.02 BOOL  ; 下右-HMI
W501.03 BOOL  ; 下左-HMI
W501.04 BOOL  ; 扫码NG料（左）
W501.05 BOOL  ; 扫码NG料（右）
W501.06 BOOL  ; 腔体有料记忆清除 hmi
W501.07 BOOL  ; 扫码记忆清除按钮
W501.08 BOOL  ; 下料拉带清料按钮
W501.09 BOOL  ; 过渡拉带记忆清除-HMI
W50.00 BOOL  ; 备用
W50.01 BOOL  ; 备用
W50.02 BOOL  ; 上料提升气缸伸出异常
W50.03 BOOL  ; 升料提升气缸缩回异常
W50.04 BOOL  ; 上左夹子闭合异常
W50.05 BOOL  ; 上左夹子张开异常
W50.06 BOOL  ; 上料右夹子闭合异常
W50.07 BOOL  ; 上右夹子张开异常
W50.08 BOOL  ; 1#合模气缸伸出异常
W50.09 BOOL  ; #1合模缩回异常
W50.10 BOOL  ; 2#合模气缸伸出异常
W50.11 BOOL  ; #2合模缩回异常
W50.12 BOOL  ; 上料升降气缸伸出异常
W50.13 BOOL  ; 升料升降气缸缩回异常
W50.14 BOOL  ; 下料提升伸出异常
W50.15 BOOL  ; 下料提升缩回异常
W510.08 BOOL  ; 空跑允许
W510.09 BOOL  ; 空跑辅助
W51.00 BOOL  ; 上料右升降气缸伸出异常
W51.01 BOOL  ; 上料升降气缸缩回异常
W51.02 BOOL  ; 下左夹闭合异常
W51.03 BOOL  ; 下左夹张开异常
W51.04 BOOL  ; 下右夹闭合异常
W51.05 BOOL  ; 下右夹张开异常
W51.06 BOOL  ; NG气缸缩回异常
W51.07 BOOL  ; NG气缸伸出异常
W51.08 BOOL  ; 上料私服异常
W51.09 BOOL  ; 下料伺服异常
W51.10 BOOL  ; 气源压力异常
W51.11 BOOL  ; 真空泵异常
W51.12 BOOL  ; 上料轴正向极限异常
W51.13 BOOL  ; 上料轴负向极限异常
W51.14 BOOL  ; 下料轴正向极限异常
W51.15 BOOL  ; 下料轴负向极限异常
W52.00 BOOL  ; 右爪上料位柔性报警
W52.01 BOOL  ; 左爪上料柔性异常
W52.02 BOOL  ; 腔体1放料柔性异常
W52.03 BOOL  ; 腔体2放料柔性异常
W52.04 BOOL  ; 下料轴2#腔体取料柔性异常
W52.05 BOOL  ; 下料轴1#腔体取料柔性异常
W52.06 BOOL  ; 下料轴右爪放ok柔性异常
W52.07 BOOL  ; 下料轴左爪放ok柔性异常
W52.08 BOOL  ; 下料轴放NG料柔性异常
W52.09 BOOL  ; 1#爪取料后上料位有料信号异常
W52.10 BOOL  ; 2爪取料后上料位有料信号异常
W52.12 BOOL  ; 柔性报警
W52.13 BOOL  ; 下料轴柔性报警
W53.00 BOOL  ; 腔体1放料后有料信号异常
W53.01 BOOL  ; 腔体1取料后有料信号异常
W53.02 BOOL  ; 腔体1无料状态跟有料信号不一致
W53.03 BOOL  ; 腔体2放料后有料信号异常
W53.04 BOOL  ; 腔体2取料后有料信号异常
W53.05 BOOL  ; 腔体2无料状态跟有料信号不一致
W53.06 BOOL  ; 上料位信号异常
W53.07 BOOL  ; 下料右爪放OK料时有料信号异常
W53.08 BOOL  ; 下料左爪放OK料有料信号异常
W53.09 BOOL  ; 前门安全开关异常
W53.10 BOOL  ; 后门安全开关异常
W53.11 BOOL  ; 左门安全开关异常
W53.12 BOOL  ; 右门安全开关异常
W53.13 BOOL  ; 急停按钮信号
W53.14 BOOL  ; 1#真空计异常
W53.15 BOOL  ; 2#真空计异常
W54.00 BOOL  ; 有料信号有料不能复位
W54.01 BOOL  ; 爪子记忆有料不能复位
W54.02 BOOL  ; 腔体有料记忆
W54.03 BOOL  ; 自动条件不满足
W54.04 BOOL  ; 氦检仪通讯异常
W54.05 BOOL  ; 氦检仪报警输出
W54.06 BOOL  ; 腔体#1有料/感应异常不能复位
W54.07 BOOL  ; 腔体#2有料/感应异常不能复位
W54.08 BOOL  ; 上料#2爪启动条件异常
W54.09 BOOL  ; 上料#2爪启动条件异常
W54.10 BOOL  ; 下料#1启动条件异常
W54.11 BOOL  ; 下料#2异常合模1缸启动条件
W54.12 BOOL  ; 合模1缸启动条件异常
W54.13 BOOL  ; 合模2缸启动条件异常
W54.14 BOOL  ; 电池流出出料拉带2超时
W54.15 BOOL  ; NG料满报警提示
W55.00 BOOL  ; NG提示
W55.01 BOOL  ; 氦检仪警报输出
W55.05 BOOL  ; TS6
W56.00 BOOL  ; 扫码位电池跟随
W5.00 BOOL  ; 真空泵-HMI
W5.01 BOOL  ; #1合模气缸-HMI
W5.02 BOOL  ; #1抽气阀-HMI
W5.03 BOOL  ; #1氦检阀-HMI
W5.04 BOOL  ; #1破真空阀-HMI
W5.05 BOOL  ; #1吹气阀-HMI
W5.06 BOOL  ; #1腔体自检-HMI
W5.07 BOOL  ; #2合模气缸-HMI
W5.08 BOOL  ; #2抽气阀-HMI
W5.09 BOOL  ; #2氦检阀-HMI
W5.10 BOOL  ; #2破真空阀-HMI
W5.11 BOOL  ; #2吹气阀-HMI
W5.12 BOOL  ; #2腔体自检-HMI
W60.00 BOOL  ; 急停触发辅助
W60.01 BOOL  ; 带料复位触发选择
W60.02 BOOL  ; 急停带料复位触发
W60.03 BOOL  ; 清料复位触发选择
W60.04 BOOL  ; 急停清料复位选择
W60.05 BOOL  ; 右位清料标志
W60.06 BOOL  ; 左位清料标志
W60.08 BOOL  ; 在1腔体标志
W60.10 BOOL  ; 右有料处理下料轴辅助
W60.11 BOOL  ; 有料复位上料轴
W60.12 BOOL  ; #2号腔体有料标志
W60.13 BOOL  ; 左有料处理下料轴辅助
W60.14 BOOL  ; #2腔体没料时辅助运行
W60.15 BOOL  ; #1腔体没料时辅助运行
W61.00 BOOL  ; 急停复位自动触发
W61.12 BOOL  ; #1号腔体有料标志
W63.13 BOOL  ; 腔体1关闭条件
W63.14 BOOL  ; 腔体1关闭条件
W64.13 BOOL  ; 合模气缸2伸出条件
W64.14 BOOL  ; 合模气缸2伸出条件
W65.01 BOOL  ; 左扫码完成
W6.00 BOOL  ; 上料机械手右爪上料位-HMI
W6.01 BOOL  ; 上料机械手腔体1位置-HMI
W6.02 BOOL  ; 上料机械手腔体2位置-HMI
W6.03 BOOL  ; 上料机械手左爪上料位-HMI
W6.04 BOOL  ; 下料右爪下OK-HMI
W6.05 BOOL  ; 下料机械手腔体1位置-HMI
W6.06 BOOL  ; 下料机械手腔体2位置-HMI
W6.07 BOOL  ; 下料机械手左OK放料位置-HMI
W6.08 BOOL  ; 下料机械手NG放料位置-HMI
W6.11 BOOL  ; 上料右扫码NG位
W6.12 BOOL  ; 上料左扫码NG位
W6.13 BOOL  ; 扫码阻挡出HMI
W7.00 BOOL  ; 电脑未启动/屏蔽
W7.02 BOOL  ; 扫码左NG HMI
W7.03 BOOL  ; 扫码右NG HMI
W7.05 BOOL  ; 忽略扫码-HMI
W7.12 BOOL  ; 再次扫码-HMI
W8.00 BOOL  ; 停止按钮-HMI
W8.01 BOOL  ; 启动按钮-HMI
W8.02 BOOL  ; 复位按钮-HMI
W8.12 BOOL  ; 上下料伺服距离过小
W8.13 BOOL  ; 进料旋转在进料反角度
W8.14 BOOL  ; 下料机械手到#1腔体安全条件
W8.15 BOOL  ; 下料机械手到#2腔体安全条件
W90.00 BOOL  ; 上料机械手在左爪上料位置
W90.01 BOOL  ; 下料轴在右爪放OK料位置
W90.06 BOOL  ; 上料轴到左爪上料位置
W91.00 BOOL  ; 上料机械手在左NG槽位置
W91.01 BOOL  ; 上料机械手在右NG槽位置
W9.00 BOOL  ; 上料机械手在右爪上料位置
W9.01 BOOL  ; 上料机械手在腔体1位置
W9.02 BOOL  ; 上料机械手在腔体2位置
W9.03 BOOL  ; 下料机械手在腔体1位置
W9.04 BOOL  ; 下料机械手在腔体2位置
W9.05 BOOL  ; 下料机械手在左爪OK放料位置
W9.06 BOOL  ; 下料机械手在NG放料位置
W9.07 BOOL  ; 进料旋转在进料1位置
W9.08 BOOL  ; 进料旋转在进料2位置
W9.09 BOOL  ; 进料旋转在上料位置
W9.10 BOOL  ; 出料旋转在出料1位置
W9.11 BOOL  ; 出料旋转在出料2位置
W9.12 BOOL  ; 出料旋转在下料位置
W9.13 BOOL  ; 机械手手动停止距离
W9.14 BOOL  ; 上料机械手到#1腔体安全条件
W9.15 BOOL  ; 上料机械手回#2腔体安全条件

## Program 程序 (cyclic task 0)
Local symbols
A DWORD
NOP BOOL
a WORD
ww40510 BOOL

### Section 起停控制

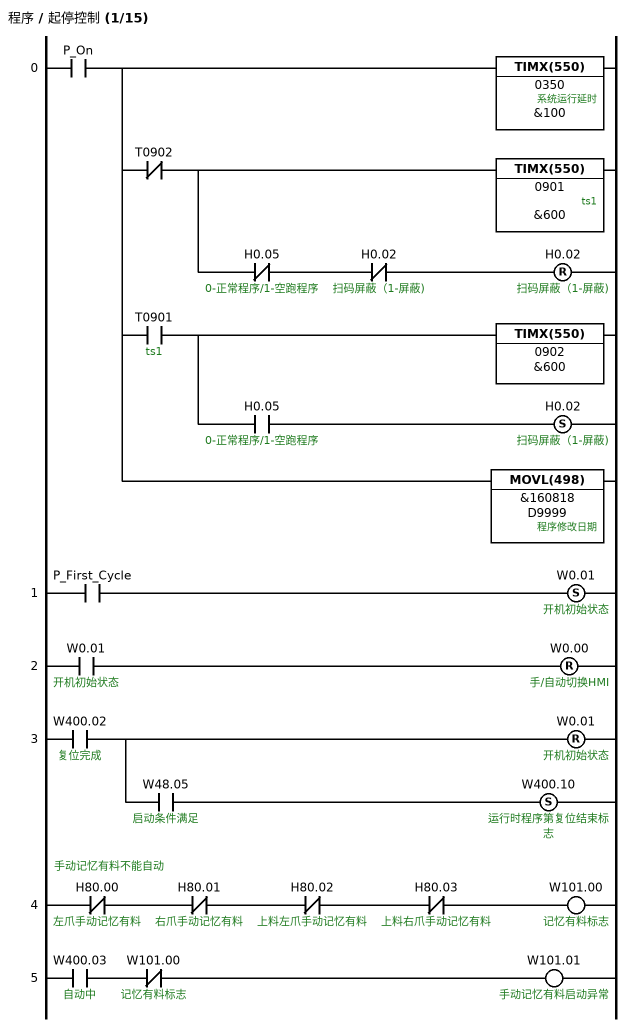
; rung 0
LD P_On
OUT TR0
TIMX(550) 0350 &100  ; 系统运行延时
ANDNOT T0902
TIMX(550) 0901 &600  ; ts1
ANDNOT H0.05  ; 0-正常程序/1-空跑程序
ANDNOT H0.02  ; 扫码屏蔽（1-屏蔽)
RSET H0.02  ; 扫码屏蔽（1-屏蔽)
LD TR0
AND T0901  ; ts1
TIMX(550) 0902 &600
AND H0.05  ; 0-正常程序/1-空跑程序
SET H0.02  ; 扫码屏蔽（1-屏蔽)
LD TR0
MOVL(498) &160818 D9999  ; 程序修改日期
; rung 1
LD P_First_Cycle
SET W0.01  ; 开机初始状态
; rung 2
LD W0.01  ; 开机初始状态
RSET W0.00  ; 手/自动切换HMI
; rung 3
LD W400.02  ; 复位完成
RSET W0.01  ; 开机初始状态
AND W48.05  ; 启动条件满足
SET W400.10  ; 运行时程序第复位结束标志
; rung 4: 手动记忆有料不能自动
LDNOT H80.00  ; 左爪手动记忆有料
ANDNOT H80.01  ; 右爪手动记忆有料
ANDNOT H80.02  ; 上料左爪手动记忆有料
ANDNOT H80.03  ; 上料右爪手动记忆有料
OUT W101.00  ; 记忆有料标志
; rung 5
LD W400.03  ; 自动中
ANDNOT W101.00  ; 记忆有料标志
OUT W101.01  ; 手动记忆有料启动异常

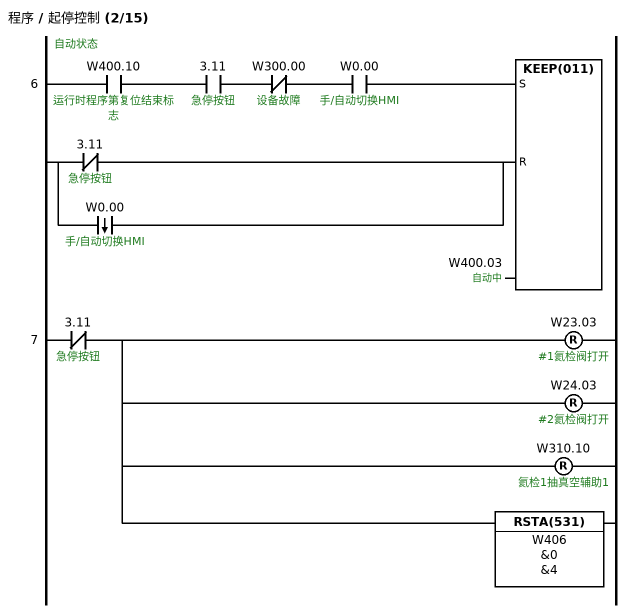
; rung 6: 自动状态
LD W400.10  ; 运行时程序第复位结束标志
AND 3.11  ; 急停按钮
ANDNOT W300.00  ; 设备故障
AND W0.00  ; 手/自动切换HMI
LDNOT 3.11  ; 急停按钮
%OR W0.00  ; 手/自动切换HMI
KEEP(011) W400.03  ; 自动中
; rung 7
LDNOT 3.11  ; 急停按钮
RSET W23.03  ; #1氦检阀打开
RSET W24.03  ; #2氦检阀打开
RSET W310.10  ; 氦检1抽真空辅助1
RSTA(531) W406 &0 &4

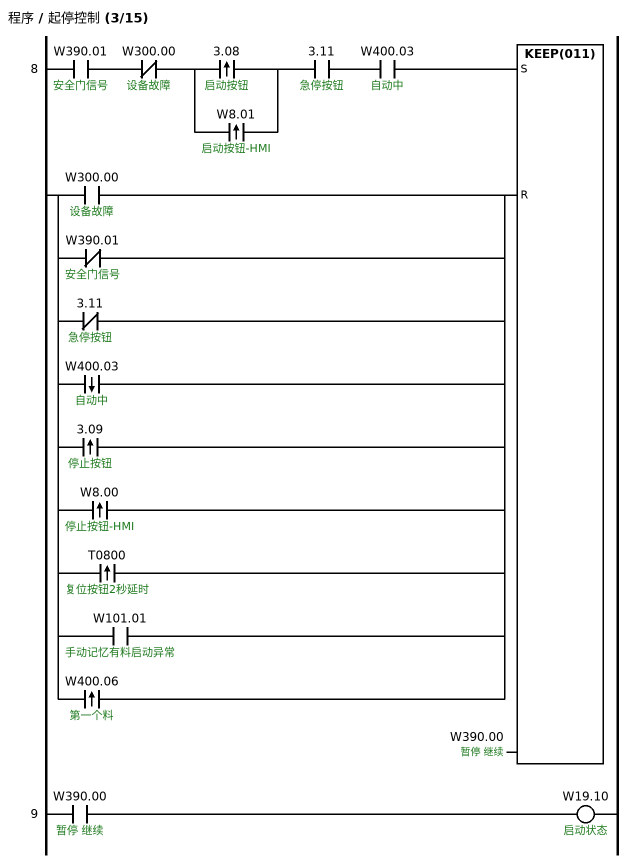
; rung 8
LD W390.01  ; 安全门信号
ANDNOT W300.00  ; 设备故障
@LD 3.08  ; 启动按钮
@OR W8.01  ; 启动按钮-HMI
ANDLD
AND 3.11  ; 急停按钮
AND W400.03  ; 自动中
LD W300.00  ; 设备故障
ORNOT W390.01  ; 安全门信号
ORNOT 3.11  ; 急停按钮
%OR W400.03  ; 自动中
@OR 3.09  ; 停止按钮
@OR W8.00  ; 停止按钮-HMI
@OR T0800  ; 复位按钮2秒延时
OR W101.01  ; 手动记忆有料启动异常
@OR W400.06  ; 第一个料
KEEP(011) W390.00  ; 暂停 继续
; rung 9
LD W390.00  ; 暂停 继续
OUT W19.10  ; 启动状态

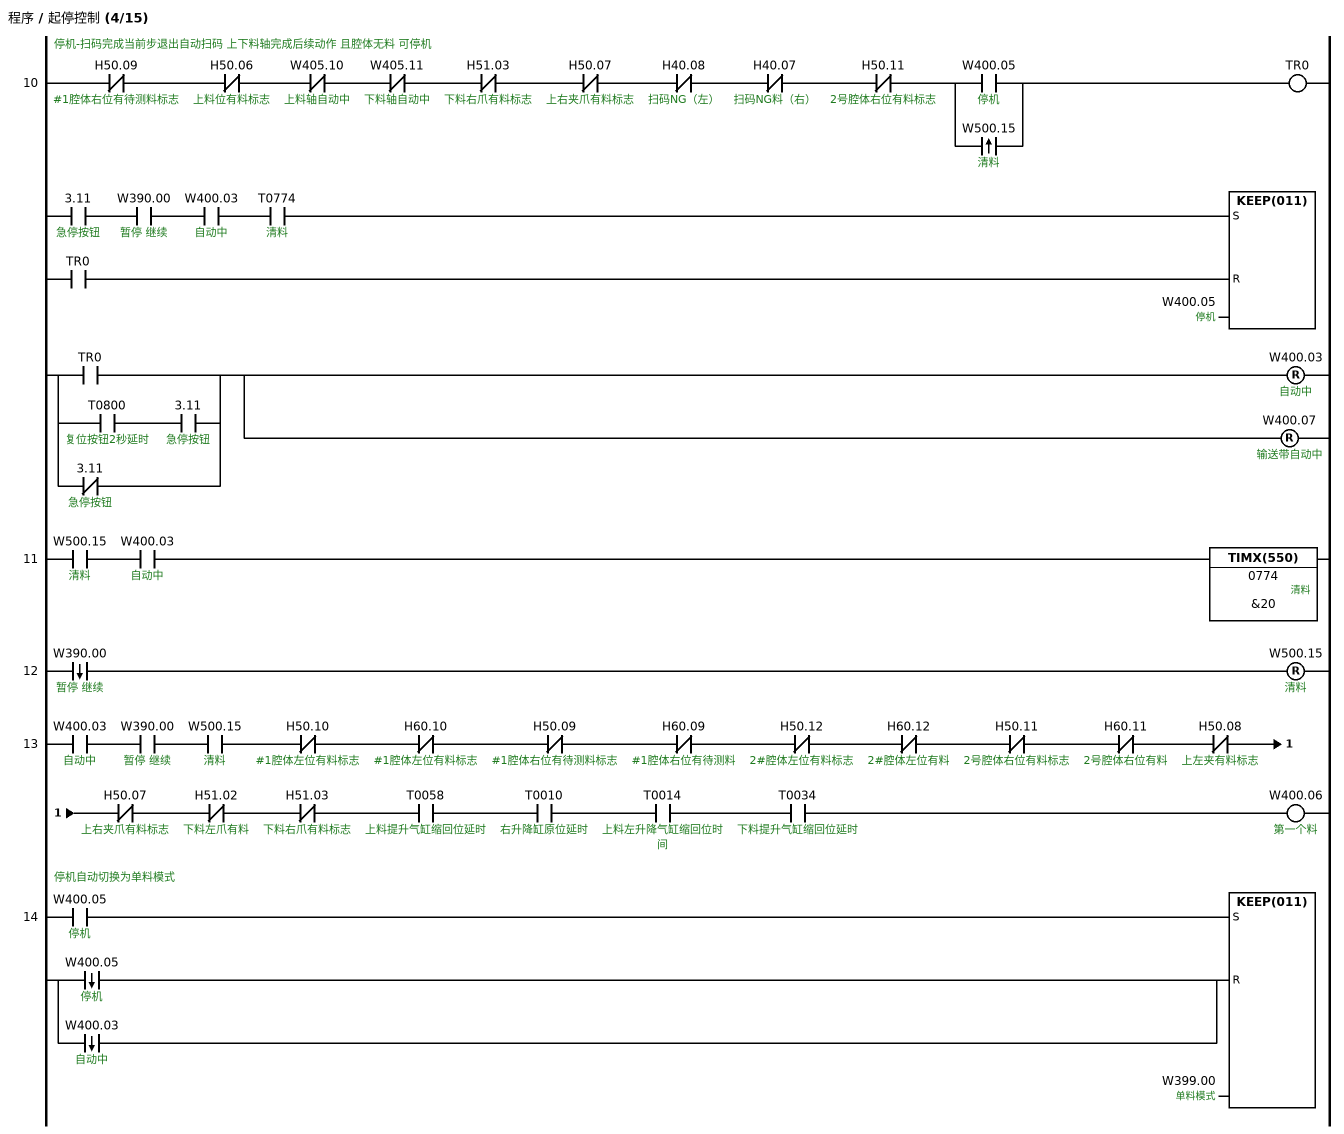
; rung 10: 停机-扫码完成当前步退出自动扫码 上下料轴完成后续动作 且腔体无料 可停机
LD 3.11  ; 急停按钮
AND W390.00  ; 暂停 继续
AND W400.03  ; 自动中
AND T0774  ; 清料
LDNOT H50.09  ; #1腔体右位有待测料标志
ANDNOT H50.06  ; 上料位有料标志
ANDNOT W405.10  ; 上料轴自动中
ANDNOT W405.11  ; 下料轴自动中
ANDNOT H51.03  ; 下料右爪有料标志
ANDNOT H50.07  ; 上右夹爪有料标志
ANDNOT H40.08  ; 扫码NG（左）
ANDNOT H40.07  ; 扫码NG料（右）
ANDNOT H50.11  ; 2号腔体右位有料标志
LD W400.05  ; 停机
@OR W500.15  ; 清料
ANDLD
OUT TR0
KEEP(011) W400.05  ; 停机
LD TR0
LD T0800  ; 复位按钮2秒延时
AND 3.11  ; 急停按钮
ORNOT 3.11  ; 急停按钮
ORLD
RSET W400.03  ; 自动中
RSET W400.07  ; 输送带自动中
; rung 11
LD W500.15  ; 清料
AND W400.03  ; 自动中
TIMX(550) 0774 &20  ; 清料
; rung 12
%LD W390.00  ; 暂停 继续
RSET W500.15  ; 清料
; rung 13
LD W400.03  ; 自动中
AND W390.00  ; 暂停 继续
AND W500.15  ; 清料
ANDNOT H50.10  ; #1腔体左位有料标志
ANDNOT H60.10  ; #1腔体左位有料标志
ANDNOT H50.09  ; #1腔体右位有待测料标志
ANDNOT H60.09  ; #1腔体右位有待测料
ANDNOT H50.12  ; 2#腔体左位有料标志
ANDNOT H60.12  ; 2#腔体左位有料
ANDNOT H50.11  ; 2号腔体右位有料标志
ANDNOT H60.11  ; 2号腔体右位有料
ANDNOT H50.08  ; 上左夹有料标志
ANDNOT H50.07  ; 上右夹爪有料标志
ANDNOT H51.02  ; 下料左爪有料
ANDNOT H51.03  ; 下料右爪有料标志
AND T0058  ; 上料提升气缸缩回位延时
AND T0010  ; 右升降缸原位延时
AND T0014  ; 上料左升降气缸缩回位时间
AND T0034  ; 下料提升气缸缩回位延时
OUT W400.06  ; 第一个料
; rung 14: 停机自动切换为单料模式
LD W400.05  ; 停机
%LD W400.05  ; 停机
%OR W400.03  ; 自动中
KEEP(011) W399.00  ; 单料模式

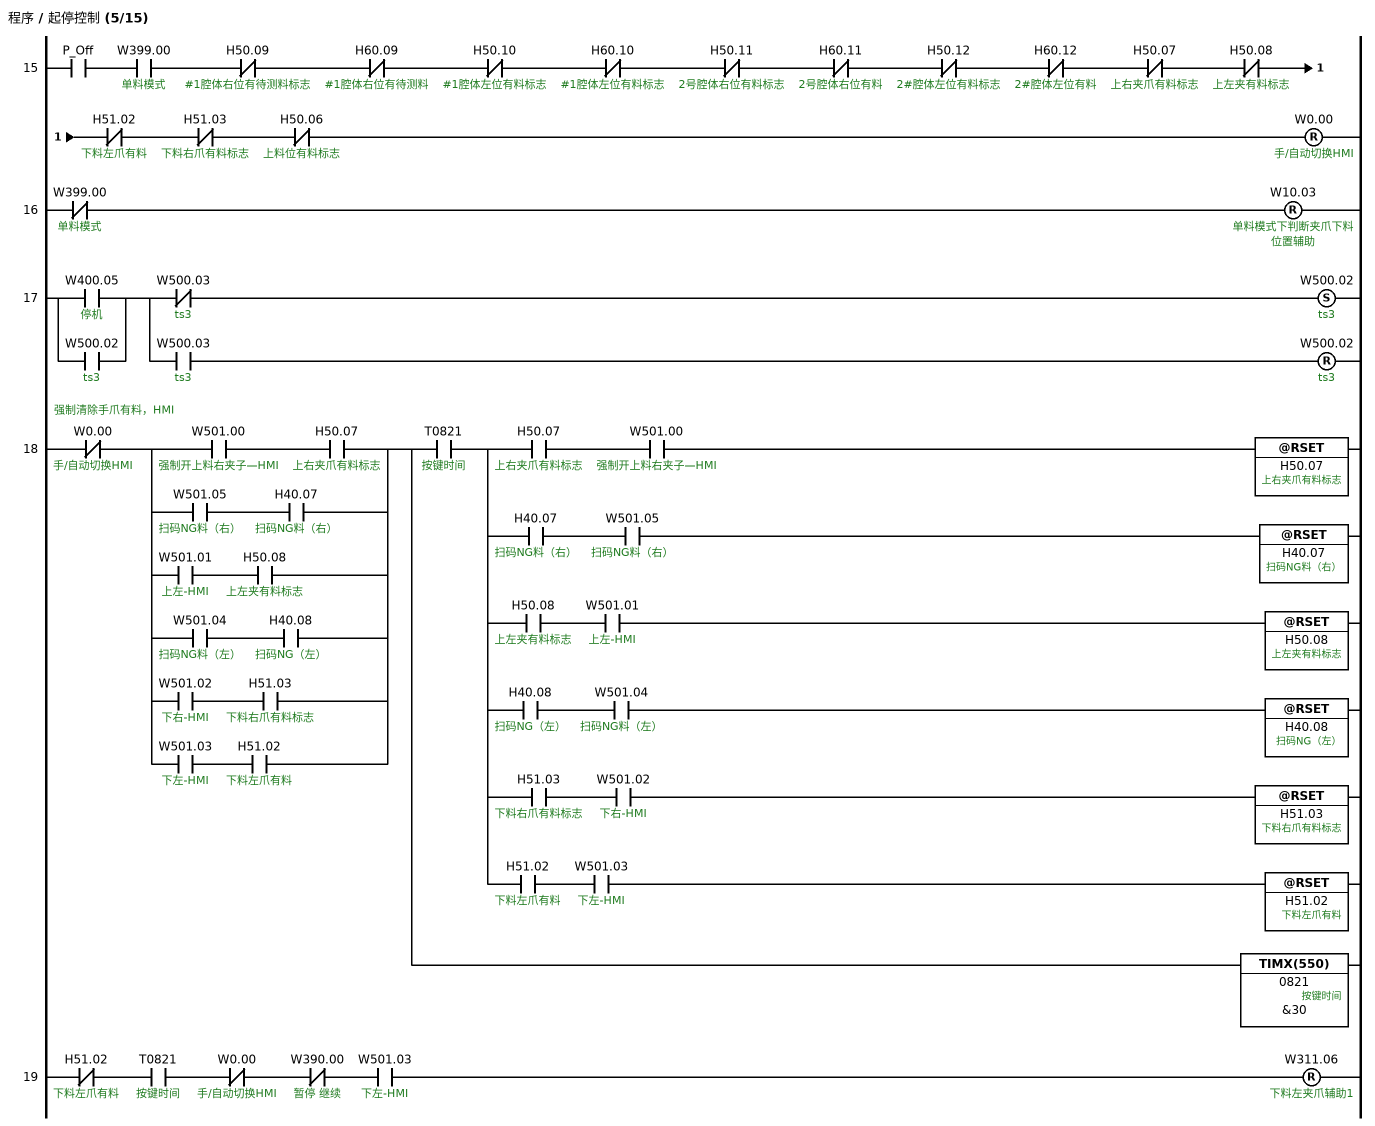
; rung 15
LD P_Off
AND W399.00  ; 单料模式
ANDNOT H50.09  ; #1腔体右位有待测料标志
ANDNOT H60.09  ; #1腔体右位有待测料
ANDNOT H50.10  ; #1腔体左位有料标志
ANDNOT H60.10  ; #1腔体左位有料标志
ANDNOT H50.11  ; 2号腔体右位有料标志
ANDNOT H60.11  ; 2号腔体右位有料
ANDNOT H50.12  ; 2#腔体左位有料标志
ANDNOT H60.12  ; 2#腔体左位有料
ANDNOT H50.07  ; 上右夹爪有料标志
ANDNOT H50.08  ; 上左夹有料标志
ANDNOT H51.02  ; 下料左爪有料
ANDNOT H51.03  ; 下料右爪有料标志
ANDNOT H50.06  ; 上料位有料标志
RSET W0.00  ; 手/自动切换HMI
; rung 16
LDNOT W399.00  ; 单料模式
RSET W10.03  ; 单料模式下判断夹爪下料位置辅助
; rung 17
LD W400.05  ; 停机
OR W500.02  ; ts3
OUT TR0
ANDNOT W500.03  ; ts3
SET W500.02  ; ts3
LD TR0
AND W500.03  ; ts3
RSET W500.02  ; ts3
; rung 18: 强制清除手爪有料，HMI
LDNOT W0.00  ; 手/自动切换HMI
LD W501.00  ; 强制开上料右夹子—HMI
AND H50.07  ; 上右夹爪有料标志
LD W501.05  ; 扫码NG料（右）
AND H40.07  ; 扫码NG料（右）
ORLD
LD W501.01  ; 上左-HMI
AND H50.08  ; 上左夹有料标志
ORLD
LD W501.04  ; 扫码NG料（左）
AND H40.08  ; 扫码NG（左）
ORLD
LD W501.02  ; 下右-HMI
AND H51.03  ; 下料右爪有料标志
ORLD
LD W501.03  ; 下左-HMI
AND H51.02  ; 下料左爪有料
ORLD
ANDLD
OUT TR0
AND T0821  ; 按键时间
OUT TR1
AND H50.07  ; 上右夹爪有料标志
AND W501.00  ; 强制开上料右夹子—HMI
@RSET H50.07  ; 上右夹爪有料标志
LD TR1
AND H40.07  ; 扫码NG料（右）
AND W501.05  ; 扫码NG料（右）
@RSET H40.07  ; 扫码NG料（右）
LD TR1
AND H50.08  ; 上左夹有料标志
AND W501.01  ; 上左-HMI
@RSET H50.08  ; 上左夹有料标志
LD TR1
AND H40.08  ; 扫码NG（左）
AND W501.04  ; 扫码NG料（左）
@RSET H40.08  ; 扫码NG（左）
LD TR1
AND H51.03  ; 下料右爪有料标志
AND W501.02  ; 下右-HMI
@RSET H51.03  ; 下料右爪有料标志
LD TR1
AND H51.02  ; 下料左爪有料
AND W501.03  ; 下左-HMI
@RSET H51.02  ; 下料左爪有料
LD TR0
TIMX(550) 0821 &30  ; 按键时间
; rung 19
LDNOT H51.02  ; 下料左爪有料
AND T0821  ; 按键时间
ANDNOT W0.00  ; 手/自动切换HMI
ANDNOT W390.00  ; 暂停 继续
AND W501.03  ; 下左-HMI
RSET W311.06  ; 下料左夹爪辅助1

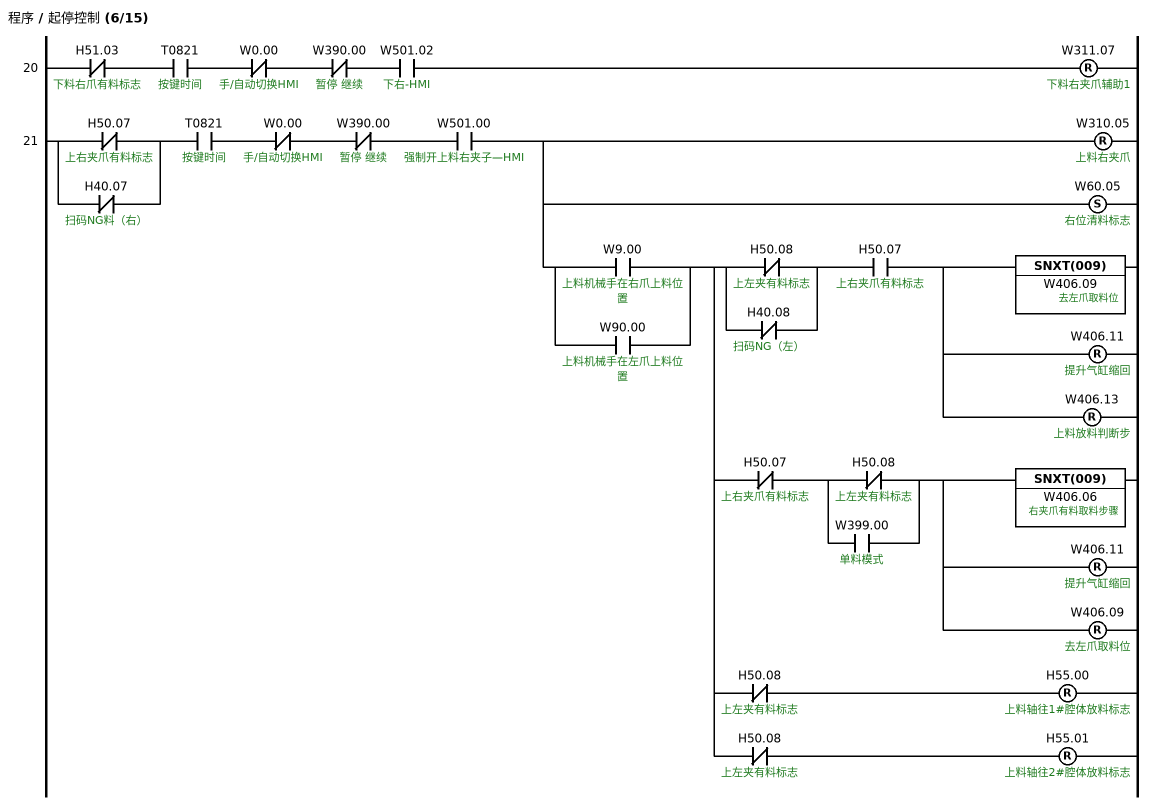
; rung 20
LDNOT H51.03  ; 下料右爪有料标志
AND T0821  ; 按键时间
ANDNOT W0.00  ; 手/自动切换HMI
ANDNOT W390.00  ; 暂停 继续
AND W501.02  ; 下右-HMI
RSET W311.07  ; 下料右夹爪辅助1
; rung 21
LDNOT H50.07  ; 上右夹爪有料标志
ORNOT H40.07  ; 扫码NG料（右）
AND T0821  ; 按键时间
ANDNOT W0.00  ; 手/自动切换HMI
ANDNOT W390.00  ; 暂停 继续
AND W501.00  ; 强制开上料右夹子—HMI
RSET W310.05  ; 上料右夹爪
SET W60.05  ; 右位清料标志
LD W9.00  ; 上料机械手在右爪上料位置
OR W90.00  ; 上料机械手在左爪上料位置
ANDLD
OUT TR0
LDNOT H50.08  ; 上左夹有料标志
ORNOT H40.08  ; 扫码NG（左）
ANDLD
AND H50.07  ; 上右夹爪有料标志
SNXT(009) W406.09  ; 去左爪取料位
RSET W406.11  ; 提升气缸缩回
RSET W406.13  ; 上料放料判断步
LD TR0
ANDNOT H50.07  ; 上右夹爪有料标志
LDNOT H50.08  ; 上左夹有料标志
OR W399.00  ; 单料模式
ANDLD
SNXT(009) W406.06  ; 右夹爪有料取料步骤
RSET W406.11  ; 提升气缸缩回
RSET W406.09  ; 去左爪取料位
LD TR0
ANDNOT H50.08  ; 上左夹有料标志
RSET H55.00  ; 上料轴往1#腔体放料标志
LD TR0
ANDNOT H50.08  ; 上左夹有料标志
RSET H55.01  ; 上料轴往2#腔体放料标志

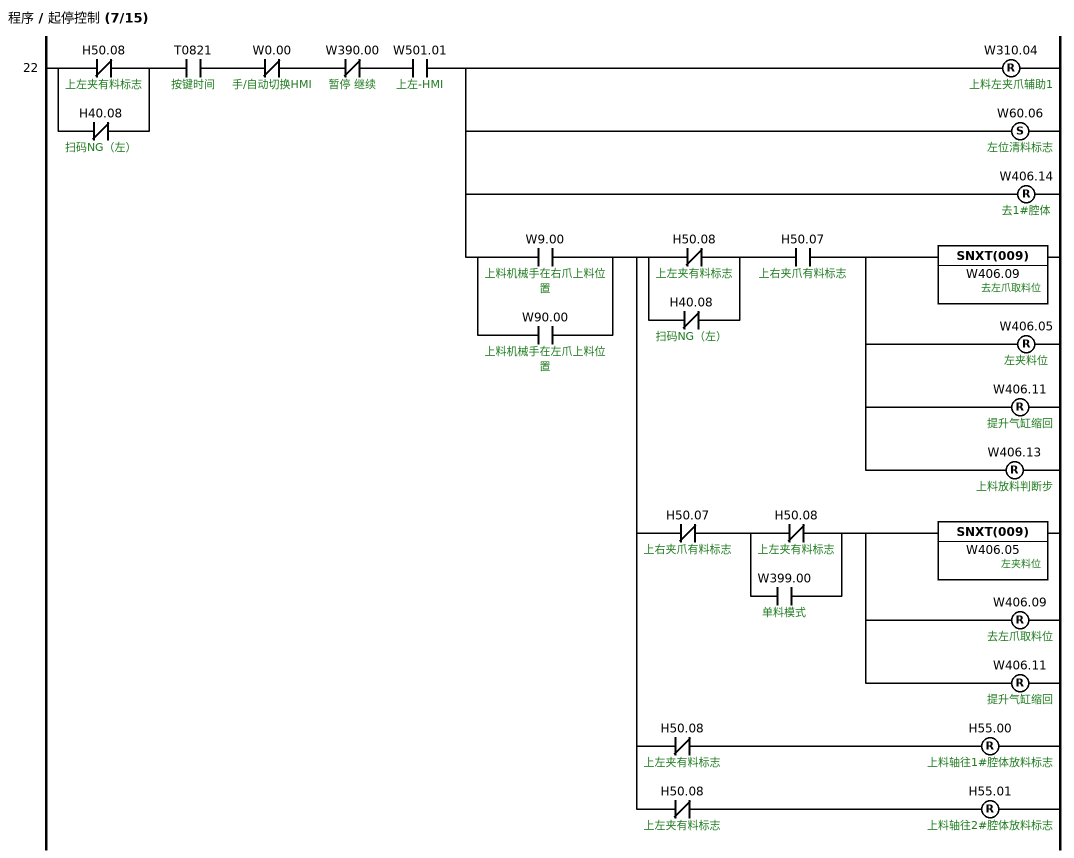
; rung 22
LDNOT H50.08  ; 上左夹有料标志
ORNOT H40.08  ; 扫码NG（左）
AND T0821  ; 按键时间
ANDNOT W0.00  ; 手/自动切换HMI
ANDNOT W390.00  ; 暂停 继续
AND W501.01  ; 上左-HMI
RSET W310.04  ; 上料左夹爪辅助1
SET W60.06  ; 左位清料标志
RSET W406.14  ; 去1#腔体
LD W9.00  ; 上料机械手在右爪上料位置
OR W90.00  ; 上料机械手在左爪上料位置
ANDLD
OUT TR0
LDNOT H50.08  ; 上左夹有料标志
ORNOT H40.08  ; 扫码NG（左）
ANDLD
AND H50.07  ; 上右夹爪有料标志
SNXT(009) W406.09  ; 去左爪取料位
RSET W406.05  ; 左夹料位
RSET W406.11  ; 提升气缸缩回
RSET W406.13  ; 上料放料判断步
LD TR0
ANDNOT H50.07  ; 上右夹爪有料标志
LDNOT H50.08  ; 上左夹有料标志
OR W399.00  ; 单料模式
ANDLD
SNXT(009) W406.05  ; 左夹料位
RSET W406.09  ; 去左爪取料位
RSET W406.11  ; 提升气缸缩回
LD TR0
ANDNOT H50.08  ; 上左夹有料标志
RSET H55.00  ; 上料轴往1#腔体放料标志
LD TR0
ANDNOT H50.08  ; 上左夹有料标志
RSET H55.01  ; 上料轴往2#腔体放料标志

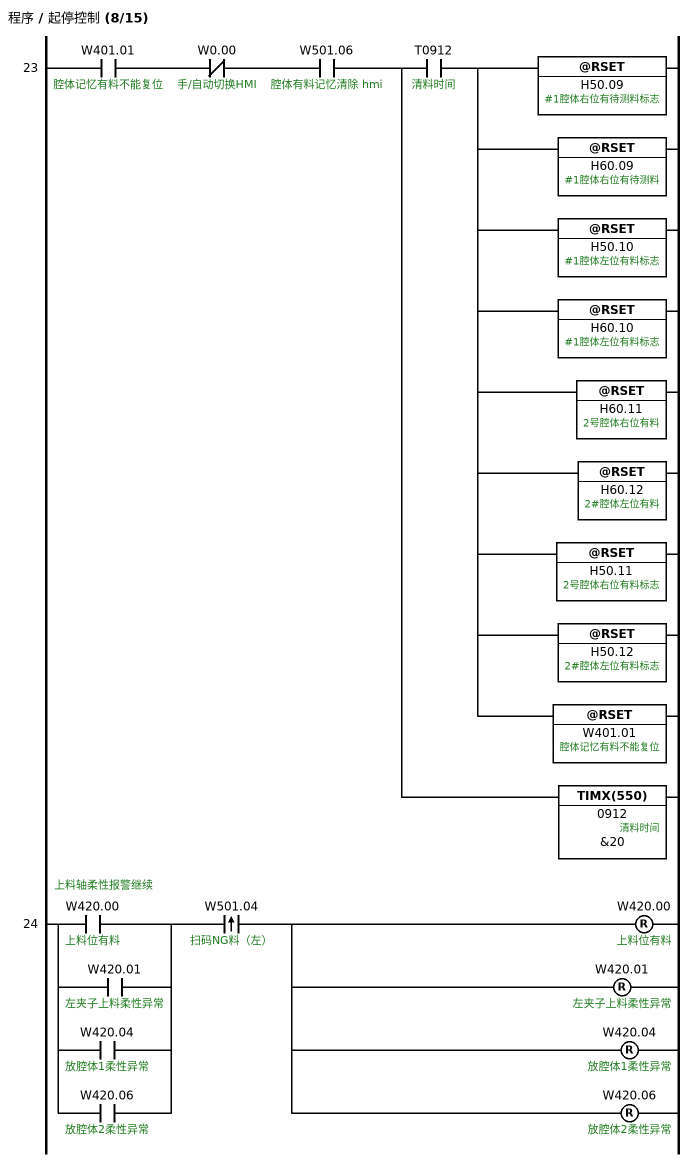
; rung 23
LD W401.01  ; 腔体记忆有料不能复位
ANDNOT W0.00  ; 手/自动切换HMI
AND W501.06  ; 腔体有料记忆清除 hmi
OUT TR0
AND T0912  ; 清料时间
@RSET H50.09  ; #1腔体右位有待测料标志
@RSET H60.09  ; #1腔体右位有待测料
@RSET H50.10  ; #1腔体左位有料标志
@RSET H60.10  ; #1腔体左位有料标志
@RSET H60.11  ; 2号腔体右位有料
@RSET H60.12  ; 2#腔体左位有料
@RSET H50.11  ; 2号腔体右位有料标志
@RSET H50.12  ; 2#腔体左位有料标志
@RSET W401.01  ; 腔体记忆有料不能复位
LD TR0
TIMX(550) 0912 &20  ; 清料时间
; rung 24: 上料轴柔性报警继续
LD W420.00  ; 上料位有料
OR W420.01  ; 左夹子上料柔性异常
OR W420.04  ; 放腔体1柔性异常
OR W420.06  ; 放腔体2柔性异常
@AND W501.04  ; 扫码NG料（左）
RSET W420.00  ; 上料位有料
RSET W420.01  ; 左夹子上料柔性异常
RSET W420.04  ; 放腔体1柔性异常
RSET W420.06  ; 放腔体2柔性异常

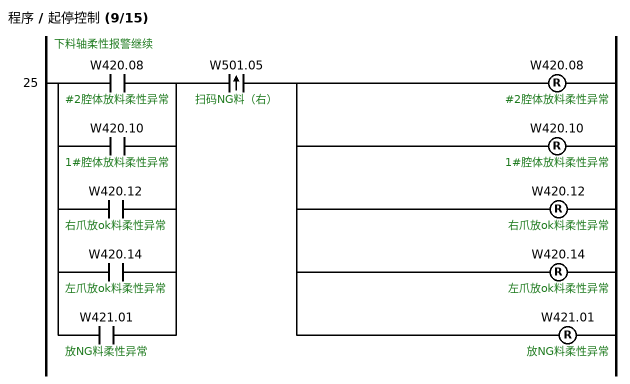
; rung 25: 下料轴柔性报警继续
LD W420.08  ; #2腔体放料柔性异常
OR W420.10  ; 1#腔体放料柔性异常
OR W420.12  ; 右爪放ok料柔性异常
OR W420.14  ; 左爪放ok料柔性异常
OR W421.01  ; 放NG料柔性异常
@AND W501.05  ; 扫码NG料（右）
RSET W420.08  ; #2腔体放料柔性异常
RSET W420.10  ; 1#腔体放料柔性异常
RSET W420.12  ; 右爪放ok料柔性异常
RSET W420.14  ; 左爪放ok料柔性异常
RSET W421.01  ; 放NG料柔性异常

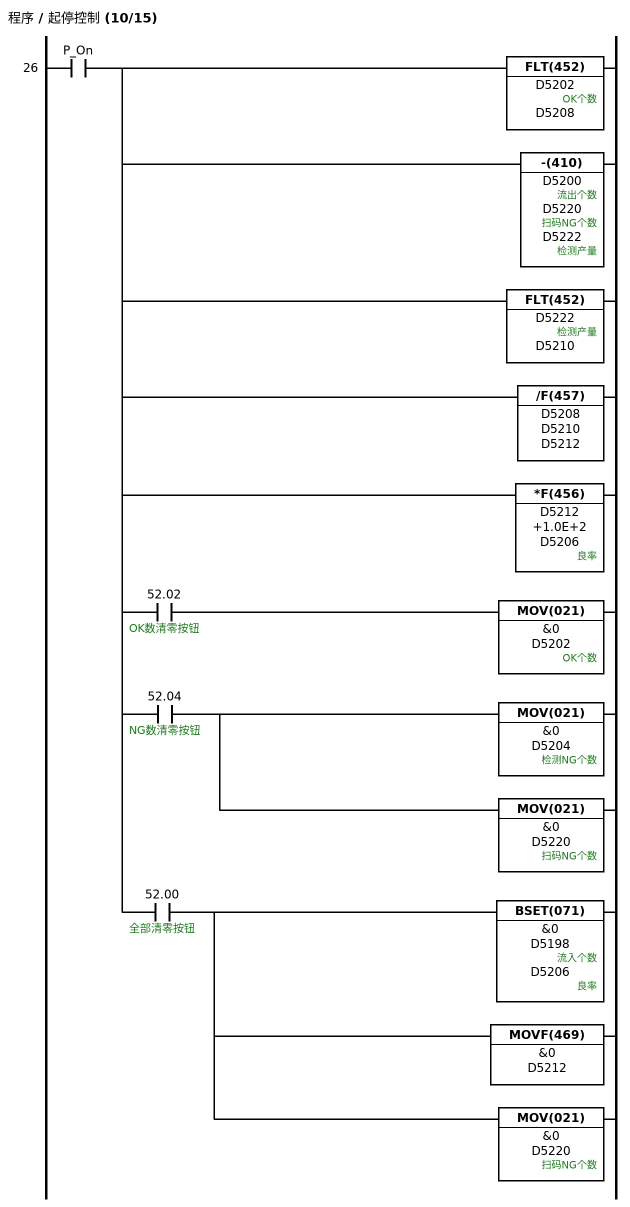
; rung 26
LD P_On
OUT TR0
FLT(452) D5202 D5208  ; OK个数
-(410) D5200 D5220 D5222  ; 流出个数, 扫码NG个数, 检测产量
FLT(452) D5222 D5210  ; 检测产量
/F(457) D5208 D5210 D5212
*F(456) D5212 +1.0E+2 D5206  ; 良率
AND 52.02  ; OK数清零按钮
MOV(021) &0 D5202  ; OK个数
LD TR0
AND 52.04  ; NG数清零按钮
MOV(021) &0 D5204  ; 检测NG个数
MOV(021) &0 D5220  ; 扫码NG个数
LD TR0
AND 52.00  ; 全部清零按钮
BSET(071) &0 D5198 D5206  ; 流入个数, 良率
MOVF(469) &0 D5212
MOV(021) &0 D5220  ; 扫码NG个数

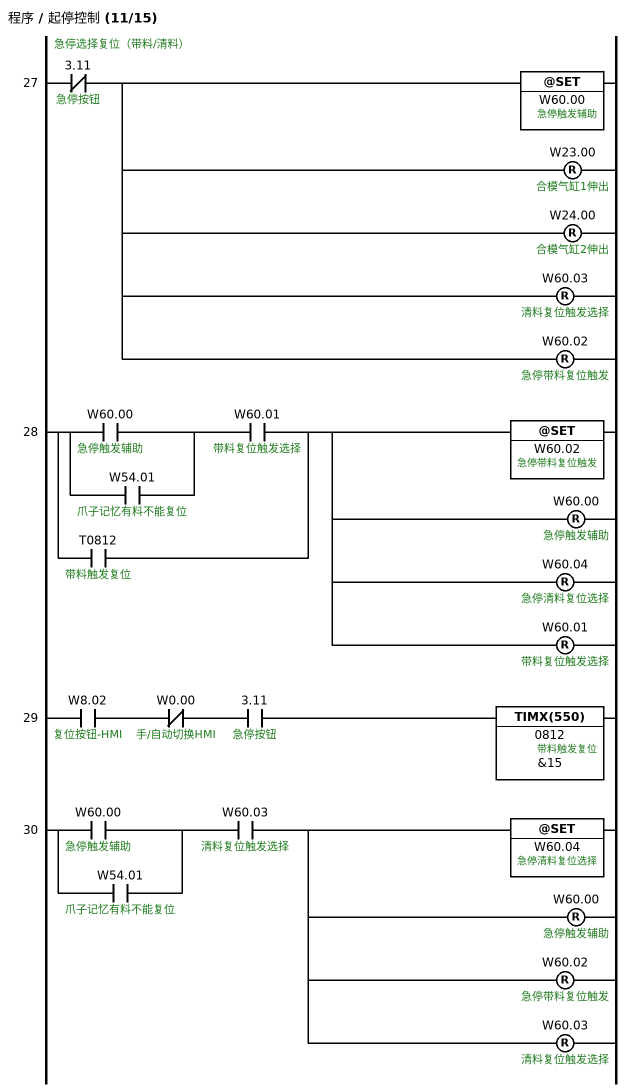
; rung 27: 急停选择复位（带料/清料）
LDNOT 3.11  ; 急停按钮
@SET W60.00  ; 急停触发辅助
RSET W23.00  ; 合模气缸1伸出
RSET W24.00  ; 合模气缸2伸出
RSET W60.03  ; 清料复位触发选择
RSET W60.02  ; 急停带料复位触发
; rung 28
LD W60.00  ; 急停触发辅助
OR W54.01  ; 爪子记忆有料不能复位
AND W60.01  ; 带料复位触发选择
OR T0812  ; 带料触发复位
@SET W60.02  ; 急停带料复位触发
RSET W60.00  ; 急停触发辅助
RSET W60.04  ; 急停清料复位选择
RSET W60.01  ; 带料复位触发选择
; rung 29
LD W8.02  ; 复位按钮-HMI
ANDNOT W0.00  ; 手/自动切换HMI
AND 3.11  ; 急停按钮
TIMX(550) 0812 &15  ; 带料触发复位
; rung 30
LD W60.00  ; 急停触发辅助
OR W54.01  ; 爪子记忆有料不能复位
AND W60.03  ; 清料复位触发选择
@SET W60.04  ; 急停清料复位选择
RSET W60.00  ; 急停触发辅助
RSET W60.02  ; 急停带料复位触发
RSET W60.03  ; 清料复位触发选择

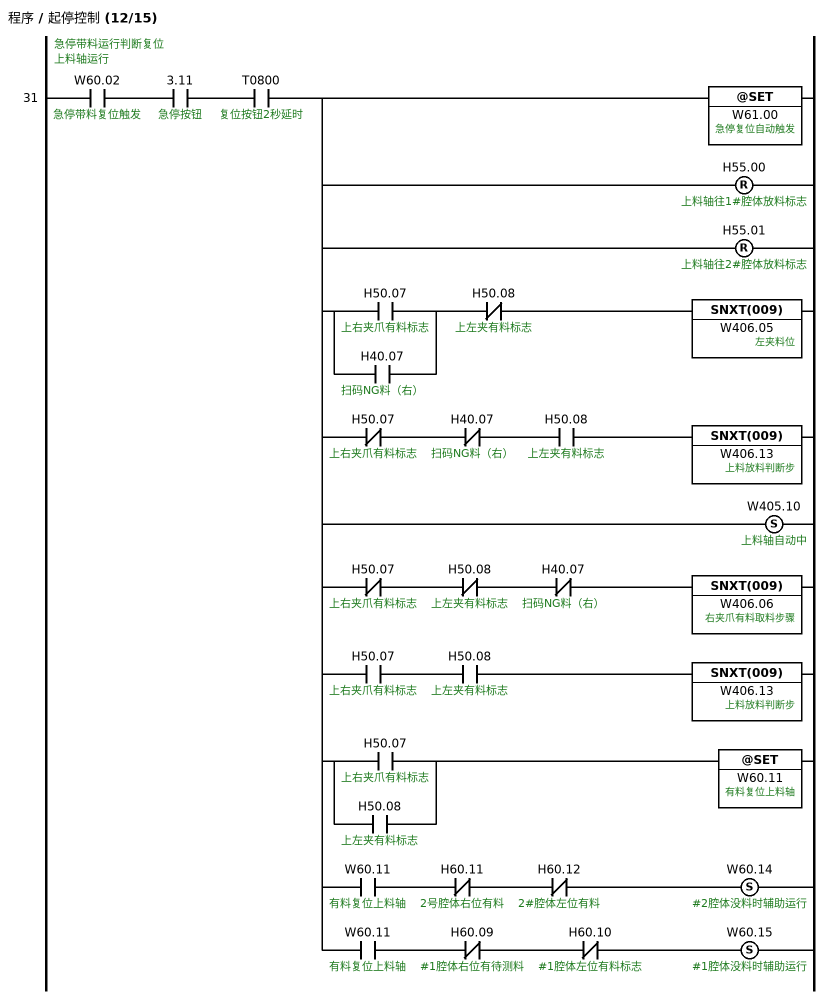
; rung 31: 急停带料运行判断复位 / 上料轴运行
LD W60.02  ; 急停带料复位触发
AND 3.11  ; 急停按钮
AND T0800  ; 复位按钮2秒延时
OUT TR0
@SET W61.00  ; 急停复位自动触发
RSET H55.00  ; 上料轴往1#腔体放料标志
RSET H55.01  ; 上料轴往2#腔体放料标志
LD H50.07  ; 上右夹爪有料标志
OR H40.07  ; 扫码NG料（右）
ANDLD
ANDNOT H50.08  ; 上左夹有料标志
SNXT(009) W406.05  ; 左夹料位
LD TR0
ANDNOT H50.07  ; 上右夹爪有料标志
ANDNOT H40.07  ; 扫码NG料（右）
AND H50.08  ; 上左夹有料标志
SNXT(009) W406.13  ; 上料放料判断步
LD TR0
SET W405.10  ; 上料轴自动中
ANDNOT H50.07  ; 上右夹爪有料标志
ANDNOT H50.08  ; 上左夹有料标志
ANDNOT H40.07  ; 扫码NG料（右）
SNXT(009) W406.06  ; 右夹爪有料取料步骤
LD TR0
AND H50.07  ; 上右夹爪有料标志
AND H50.08  ; 上左夹有料标志
SNXT(009) W406.13  ; 上料放料判断步
LD TR0
LD H50.07  ; 上右夹爪有料标志
OR H50.08  ; 上左夹有料标志
ANDLD
@SET W60.11  ; 有料复位上料轴
LD TR0
AND W60.11  ; 有料复位上料轴
ANDNOT H60.11  ; 2号腔体右位有料
ANDNOT H60.12  ; 2#腔体左位有料
SET W60.14  ; #2腔体没料时辅助运行
LD TR0
AND W60.11  ; 有料复位上料轴
ANDNOT H60.09  ; #1腔体右位有待测料
ANDNOT H60.10  ; #1腔体左位有料标志
SET W60.15  ; #1腔体没料时辅助运行

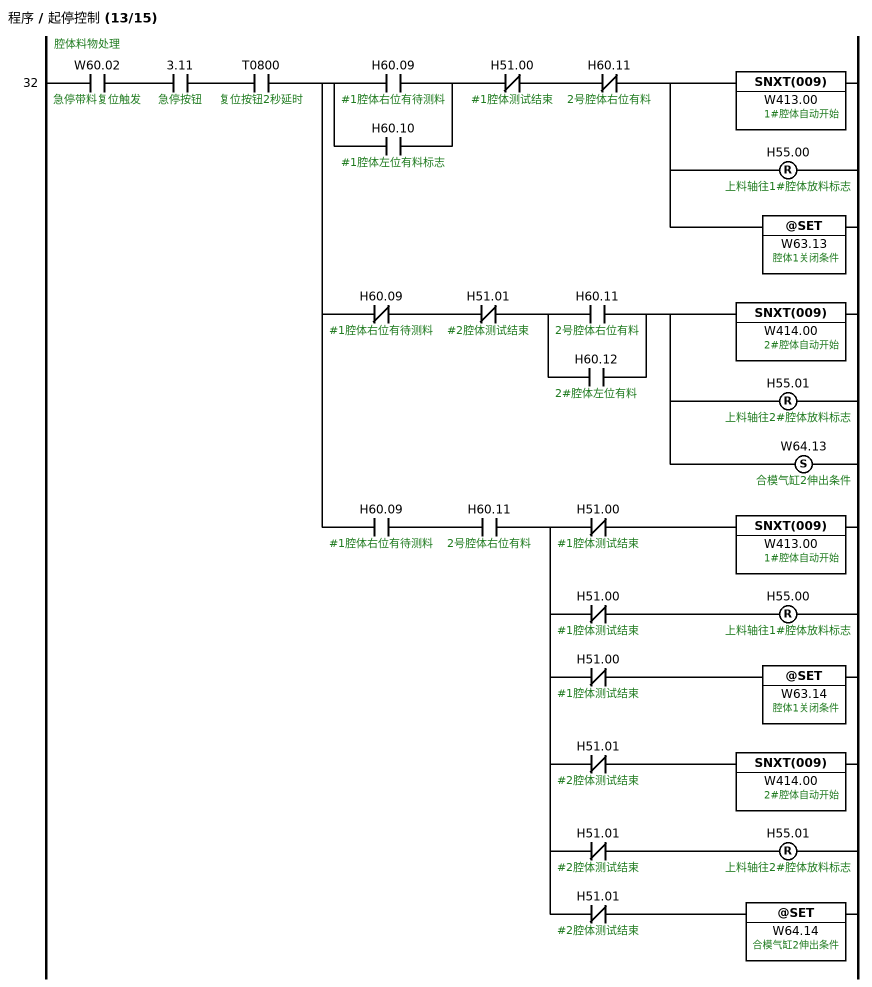
; rung 32: 腔体料物处理
LD W60.02  ; 急停带料复位触发
AND 3.11  ; 急停按钮
AND T0800  ; 复位按钮2秒延时
OUT TR0
LD H60.09  ; #1腔体右位有待测料
OR H60.10  ; #1腔体左位有料标志
ANDLD
ANDNOT H51.00  ; #1腔体测试结束
ANDNOT H60.11  ; 2号腔体右位有料
SNXT(009) W413.00  ; 1#腔体自动开始
RSET H55.00  ; 上料轴往1#腔体放料标志
@SET W63.13  ; 腔体1关闭条件
LD TR0
ANDNOT H60.09  ; #1腔体右位有待测料
ANDNOT H51.01  ; #2腔体测试结束
LD H60.11  ; 2号腔体右位有料
OR H60.12  ; 2#腔体左位有料
ANDLD
SNXT(009) W414.00  ; 2#腔体自动开始
RSET H55.01  ; 上料轴往2#腔体放料标志
SET W64.13  ; 合模气缸2伸出条件
LD TR0
AND H60.09  ; #1腔体右位有待测料
AND H60.11  ; 2号腔体右位有料
OUT TR0
ANDNOT H51.00  ; #1腔体测试结束
SNXT(009) W413.00  ; 1#腔体自动开始
LD TR0
ANDNOT H51.00  ; #1腔体测试结束
RSET H55.00  ; 上料轴往1#腔体放料标志
LD TR0
ANDNOT H51.00  ; #1腔体测试结束
@SET W63.14  ; 腔体1关闭条件
LD TR0
ANDNOT H51.01  ; #2腔体测试结束
SNXT(009) W414.00  ; 2#腔体自动开始
LD TR0
ANDNOT H51.01  ; #2腔体测试结束
RSET H55.01  ; 上料轴往2#腔体放料标志
LD TR0
ANDNOT H51.01  ; #2腔体测试结束
@SET W64.14  ; 合模气缸2伸出条件

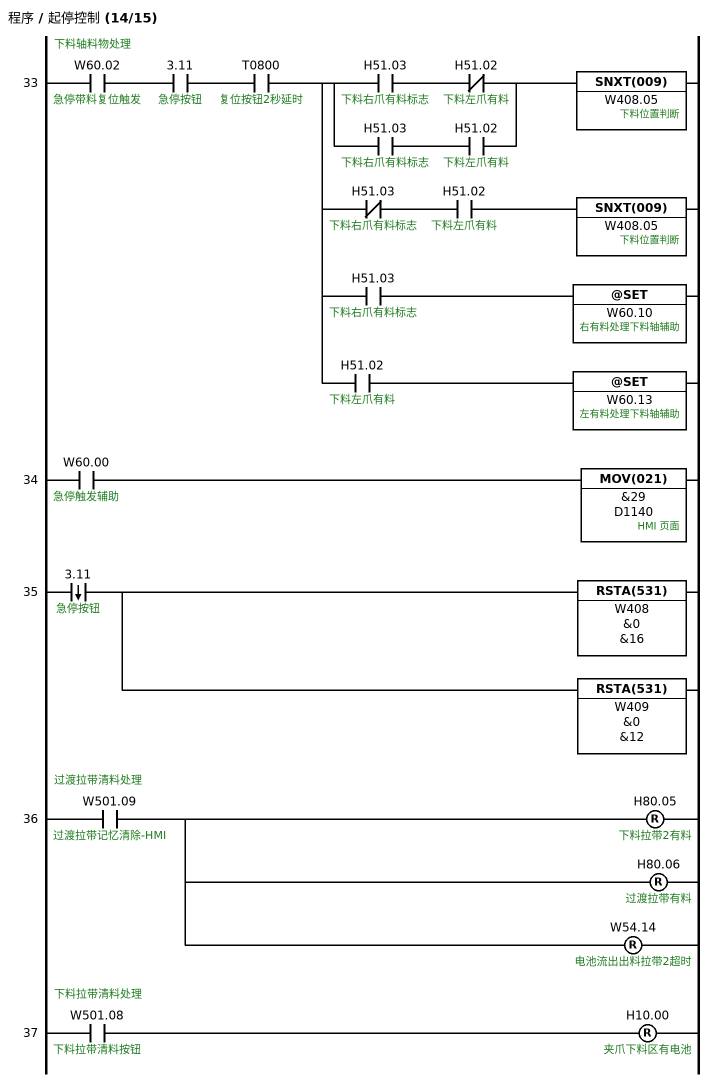
; rung 33: 下料轴料物处理
LD W60.02  ; 急停带料复位触发
AND 3.11  ; 急停按钮
AND T0800  ; 复位按钮2秒延时
OUT TR0
LD H51.03  ; 下料右爪有料标志
ANDNOT H51.02  ; 下料左爪有料
LD H51.03  ; 下料右爪有料标志
AND H51.02  ; 下料左爪有料
ORLD
ANDLD
SNXT(009) W408.05  ; 下料位置判断
LD TR0
ANDNOT H51.03  ; 下料右爪有料标志
AND H51.02  ; 下料左爪有料
SNXT(009) W408.05  ; 下料位置判断
LD TR0
AND H51.03  ; 下料右爪有料标志
@SET W60.10  ; 右有料处理下料轴辅助
LD TR0
AND H51.02  ; 下料左爪有料
@SET W60.13  ; 左有料处理下料轴辅助
; rung 34
LD W60.00  ; 急停触发辅助
MOV(021) &29 D1140  ; HMI 页面
; rung 35
%LD 3.11  ; 急停按钮
RSTA(531) W408 &0 &16
RSTA(531) W409 &0 &12
; rung 36: 过渡拉带清料处理
LD W501.09  ; 过渡拉带记忆清除-HMI
RSET H80.05  ; 下料拉带2有料
RSET H80.06  ; 过渡拉带有料
RSET W54.14  ; 电池流出出料拉带2超时
; rung 37: 下料拉带清料处理
LD W501.08  ; 下料拉带清料按钮
RSET H10.00  ; 夹爪下料区有电池

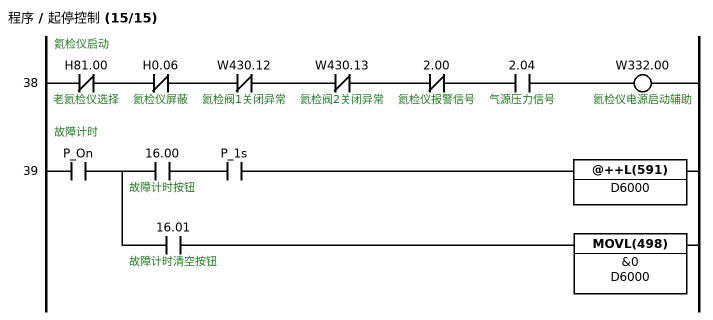
; rung 38: 氦检仪启动
LDNOT H81.00  ; 老氦检仪选择
ANDNOT H0.06  ; 氦检仪屏蔽
ANDNOT W430.12  ; 氦检阀1关闭异常
ANDNOT W430.13  ; 氦检阀2关闭异常
ANDNOT 2.00  ; 氦检仪报警信号
AND 2.04  ; 气源压力信号
OUT W332.00  ; 氦检仪电源启动辅助
; rung 39: 故障计时
LD P_On
OUT TR0
AND 16.00  ; 故障计时按钮
AND P_1s
@++L(591) D6000
LD TR0
AND 16.01  ; 故障计时清空按钮
MOVL(498) &0 D6000

### Section 复位

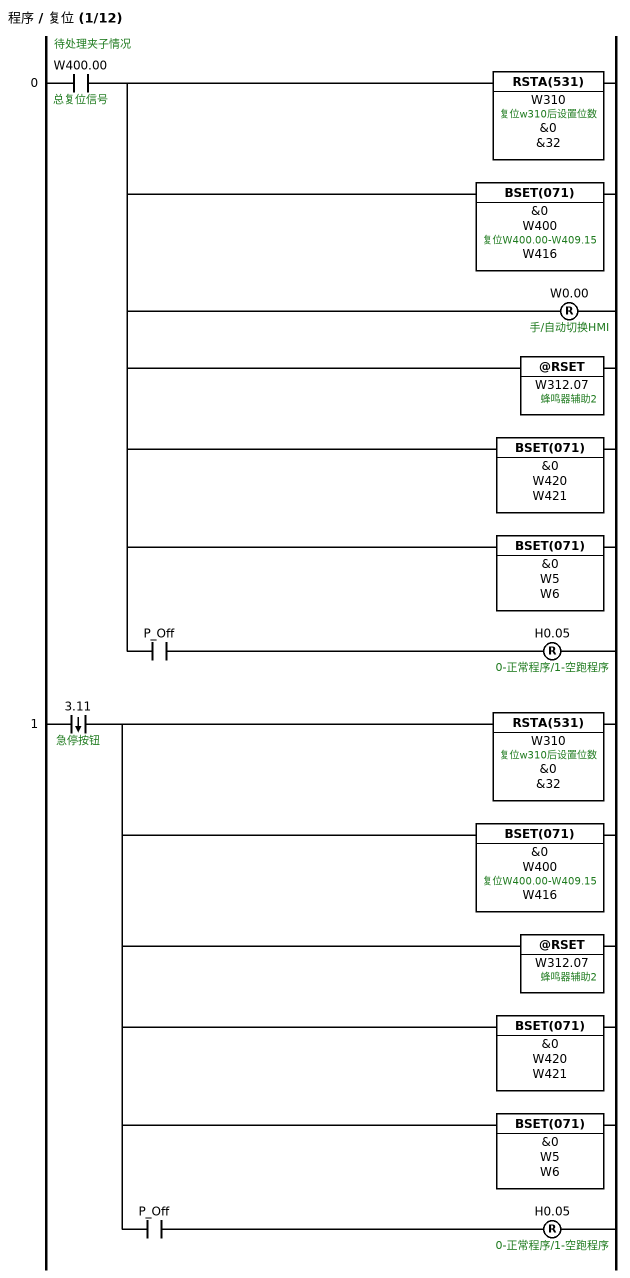
; rung 0: 待处理夹子情况
LD W400.00  ; 总复位信号
RSTA(531) W310 &0 &32  ; 复位w310后设置位数
BSET(071) &0 W400 W416  ; 复位W400.00-W409.15
RSET W0.00  ; 手/自动切换HMI
@RSET W312.07  ; 蜂鸣器辅助2
BSET(071) &0 W420 W421
BSET(071) &0 W5 W6
AND P_Off
RSET H0.05  ; 0-正常程序/1-空跑程序
; rung 1
%LD 3.11  ; 急停按钮
RSTA(531) W310 &0 &32  ; 复位w310后设置位数
BSET(071) &0 W400 W416  ; 复位W400.00-W409.15
@RSET W312.07  ; 蜂鸣器辅助2
BSET(071) &0 W420 W421
BSET(071) &0 W5 W6
AND P_Off
RSET H0.05  ; 0-正常程序/1-空跑程序

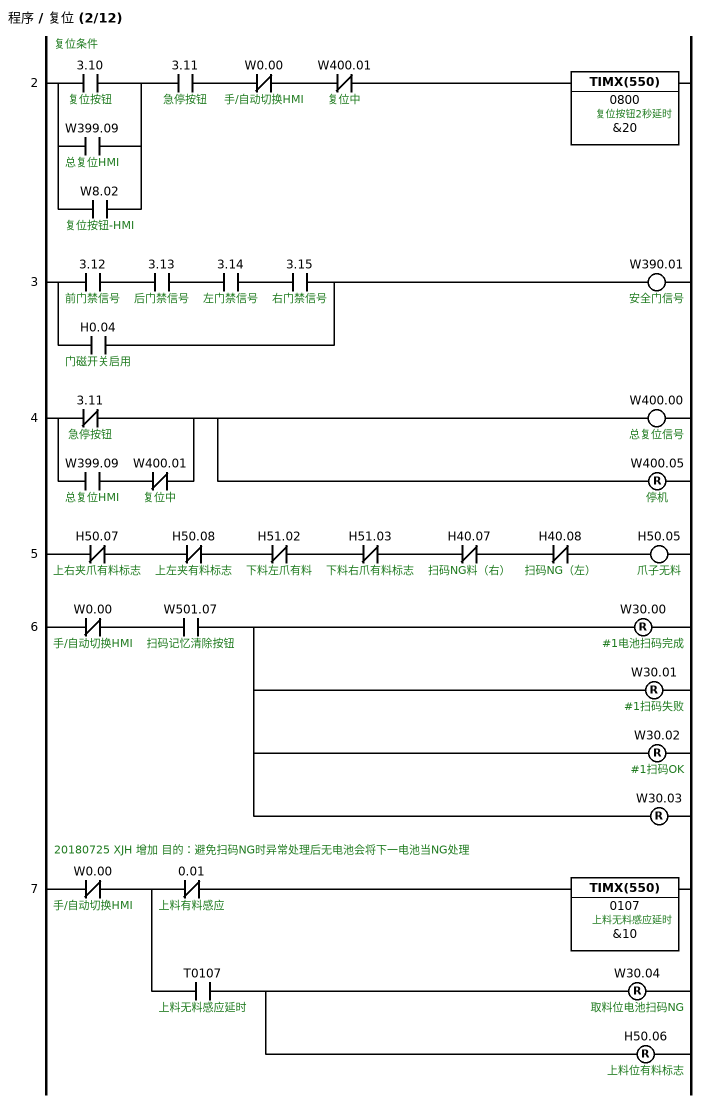
; rung 2: 复位条件
LD 3.10  ; 复位按钮
OR W399.09  ; 总复位HMI
OR W8.02  ; 复位按钮-HMI
AND 3.11  ; 急停按钮
ANDNOT W0.00  ; 手/自动切换HMI
ANDNOT W400.01  ; 复位中
TIMX(550) 0800 &20  ; 复位按钮2秒延时
; rung 3
LD 3.12  ; 前门禁信号
AND 3.13  ; 后门禁信号
AND 3.14  ; 左门禁信号
AND 3.15  ; 右门禁信号
OR H0.04  ; 门磁开关启用
OUT W390.01  ; 安全门信号
; rung 4
LDNOT 3.11  ; 急停按钮
LD W399.09  ; 总复位HMI
ANDNOT W400.01  ; 复位中
ORLD
OUT W400.00  ; 总复位信号
RSET W400.05  ; 停机
; rung 5
LDNOT H50.07  ; 上右夹爪有料标志
ANDNOT H50.08  ; 上左夹有料标志
ANDNOT H51.02  ; 下料左爪有料
ANDNOT H51.03  ; 下料右爪有料标志
ANDNOT H40.07  ; 扫码NG料（右）
ANDNOT H40.08  ; 扫码NG（左）
OUT H50.05  ; 爪子无料
; rung 6
LDNOT W0.00  ; 手/自动切换HMI
AND W501.07  ; 扫码记忆清除按钮
RSET W30.00  ; #1电池扫码完成
RSET W30.01  ; #1扫码失败
RSET W30.02  ; #1扫码OK
RSET W30.03
; rung 7: 20180725 XJH 增加 目的：避免扫码NG时异常处理后无电池会将下一电池当NG处理
LDNOT W0.00  ; 手/自动切换HMI
OUT TR0
ANDNOT 0.01  ; 上料有料感应
TIMX(550) 0107 &10  ; 上料无料感应延时
LD TR0
AND T0107  ; 上料无料感应延时
RSET W30.04  ; 取料位电池扫码NG
RSET H50.06  ; 上料位有料标志

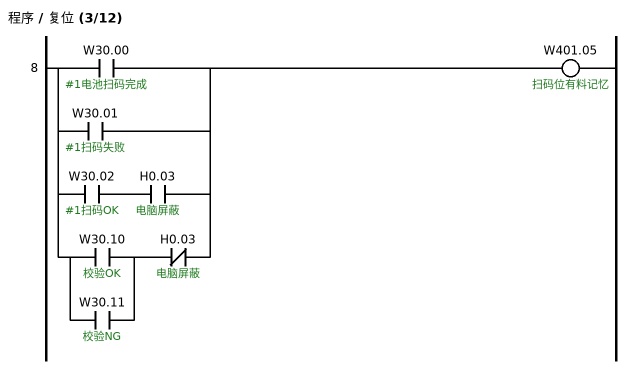
; rung 8
LD W30.00  ; #1电池扫码完成
OR W30.01  ; #1扫码失败
LD W30.02  ; #1扫码OK
AND H0.03  ; 电脑屏蔽
ORLD
LD W30.10  ; 校验OK
OR W30.11  ; 校验NG
ANDNOT H0.03  ; 电脑屏蔽
ORLD
OUT W401.05  ; 扫码位有料记忆

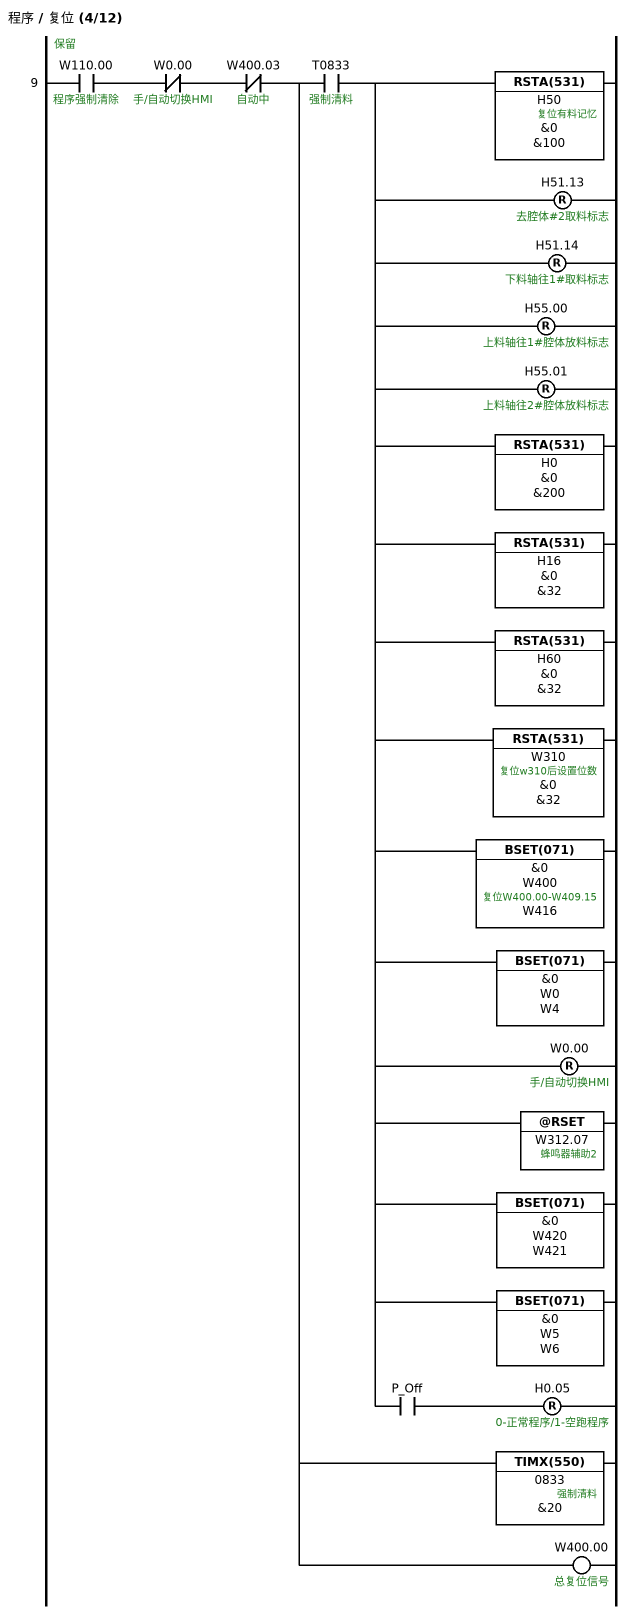
; rung 9: 保留
LD W110.00  ; 程序强制清除
ANDNOT W0.00  ; 手/自动切换HMI
ANDNOT W400.03  ; 自动中
OUT TR0
AND T0833  ; 强制清料
RSTA(531) H50 &0 &100  ; 复位有料记忆
RSET H51.13  ; 去腔体#2取料标志
RSET H51.14  ; 下料轴往1#取料标志
RSET H55.00  ; 上料轴往1#腔体放料标志
RSET H55.01  ; 上料轴往2#腔体放料标志
RSTA(531) H0 &0 &200
RSTA(531) H16 &0 &32
RSTA(531) H60 &0 &32
RSTA(531) W310 &0 &32  ; 复位w310后设置位数
BSET(071) &0 W400 W416  ; 复位W400.00-W409.15
BSET(071) &0 W0 W4
RSET W0.00  ; 手/自动切换HMI
@RSET W312.07  ; 蜂鸣器辅助2
BSET(071) &0 W420 W421
BSET(071) &0 W5 W6
AND P_Off
RSET H0.05  ; 0-正常程序/1-空跑程序
LD TR0
TIMX(550) 0833 &20  ; 强制清料
OUT W400.00  ; 总复位信号

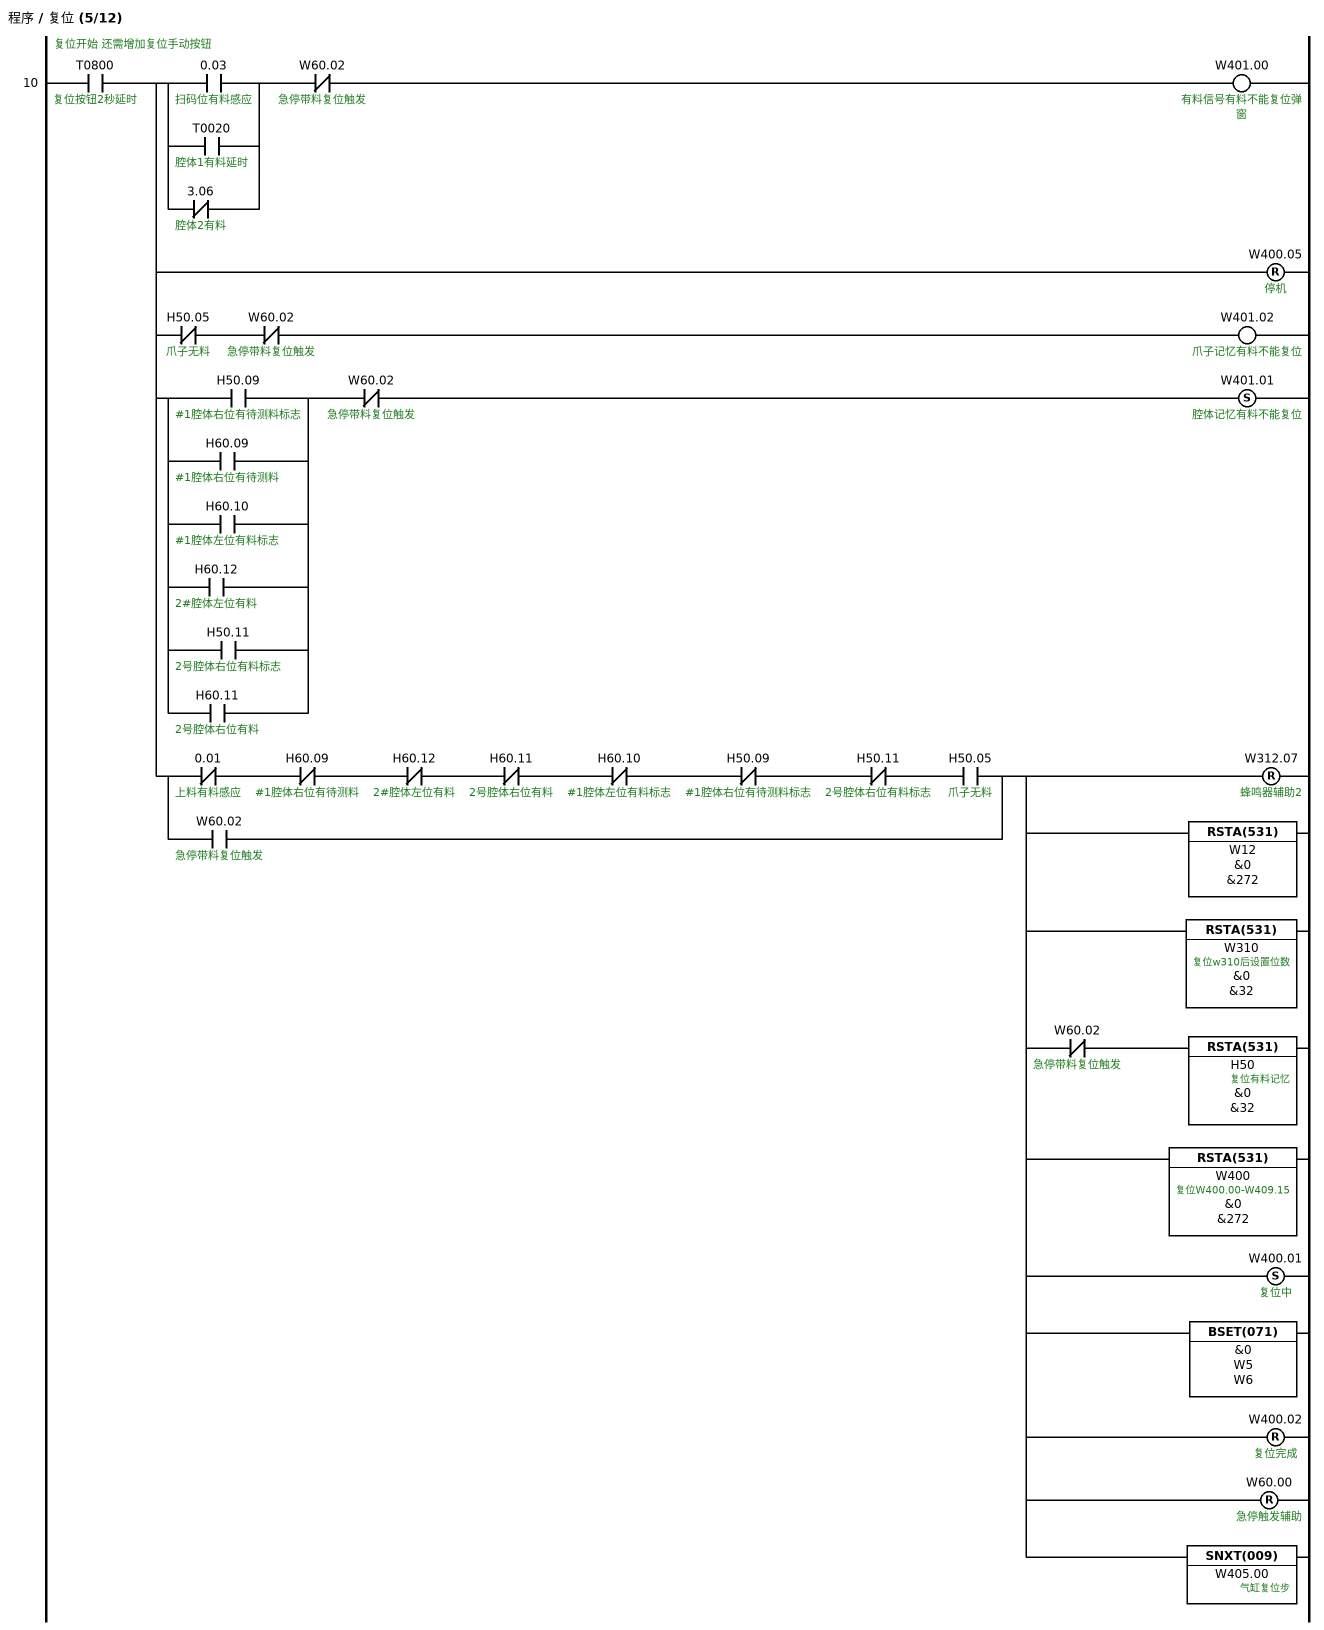
; rung 10: 复位开始 还需增加复位手动按钮
LD T0800  ; 复位按钮2秒延时
OUT TR0
LD 0.03  ; 扫码位有料感应
OR T0020  ; 腔体1有料延时
ORNOT 3.06  ; 腔体2有料
ANDLD
ANDNOT W60.02  ; 急停带料复位触发
OUT W401.00  ; 有料信号有料不能复位弹窗
LD TR0
RSET W400.05  ; 停机
ANDNOT H50.05  ; 爪子无料
ANDNOT W60.02  ; 急停带料复位触发
OUT W401.02  ; 爪子记忆有料不能复位
LD TR0
LD H50.09  ; #1腔体右位有待测料标志
OR H60.09  ; #1腔体右位有待测料
OR H60.10  ; #1腔体左位有料标志
OR H60.12  ; 2#腔体左位有料
OR H50.11  ; 2号腔体右位有料标志
OR H60.11  ; 2号腔体右位有料
ANDLD
ANDNOT W60.02  ; 急停带料复位触发
SET W401.01  ; 腔体记忆有料不能复位
LD TR0
LDNOT 0.01  ; 上料有料感应
ANDNOT H60.09  ; #1腔体右位有待测料
ANDNOT H60.12  ; 2#腔体左位有料
ANDNOT H60.11  ; 2号腔体右位有料
ANDNOT H60.10  ; #1腔体左位有料标志
ANDNOT H50.09  ; #1腔体右位有待测料标志
ANDNOT H50.11  ; 2号腔体右位有料标志
AND H50.05  ; 爪子无料
OR W60.02  ; 急停带料复位触发
ANDLD
OUT TR0
RSET W312.07  ; 蜂鸣器辅助2
RSTA(531) W12 &0 &272
RSTA(531) W310 &0 &32  ; 复位w310后设置位数
ANDNOT W60.02  ; 急停带料复位触发
RSTA(531) H50 &0 &32  ; 复位有料记忆
LD TR0
RSTA(531) W400 &0 &272  ; 复位W400.00-W409.15
SET W400.01  ; 复位中
BSET(071) &0 W5 W6
RSET W400.02  ; 复位完成
RSET W60.00  ; 急停触发辅助
SNXT(009) W405.00  ; 气缸复位步

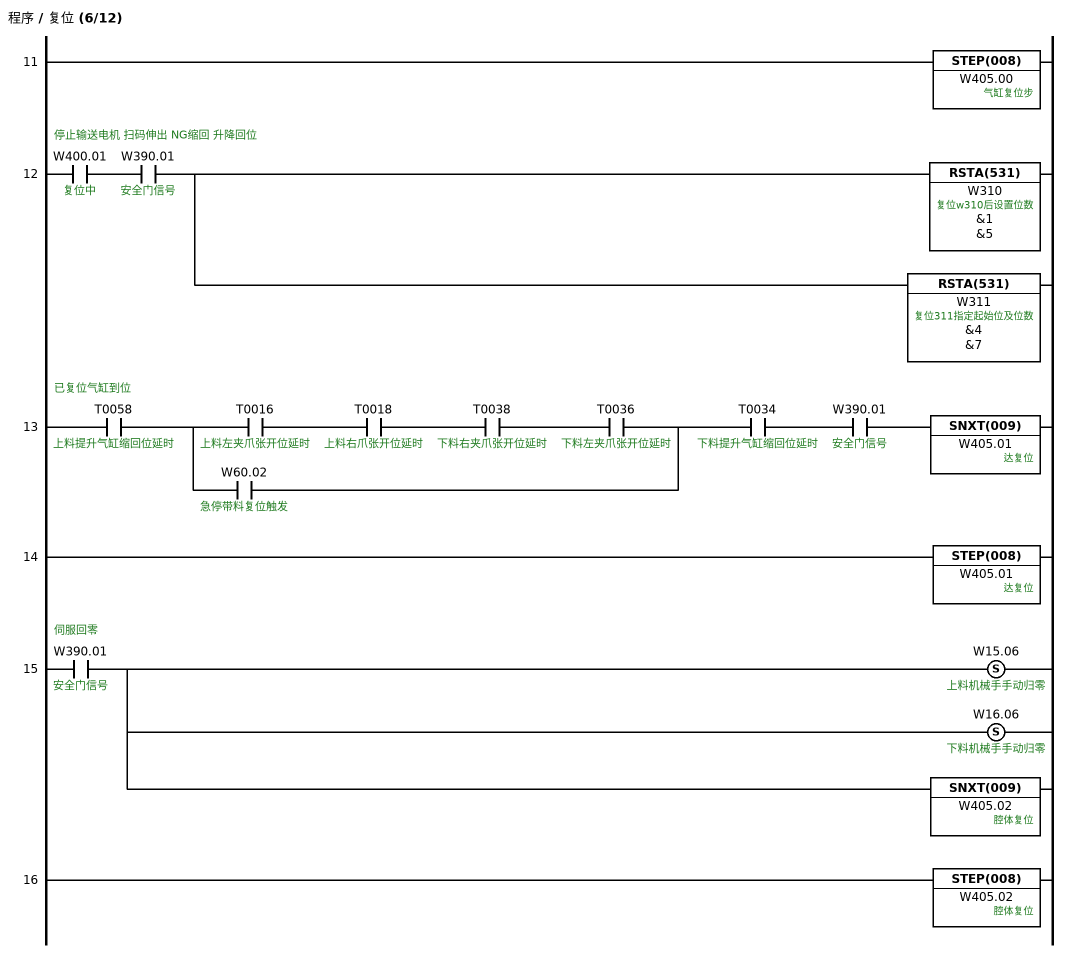
; rung 11
STEP(008) W405.00  ; 气缸复位步
; rung 12: 停止输送电机 扫码伸出 NG缩回 升降回位
LD W400.01  ; 复位中
AND W390.01  ; 安全门信号
RSTA(531) W310 &1 &5  ; 复位w310后设置位数
RSTA(531) W311 &4 &7  ; 复位311指定起始位及位数
; rung 13: 已复位气缸到位
LD T0058  ; 上料提升气缸缩回位延时
LD T0016  ; 上料左夹爪张开位延时
AND T0018  ; 上料右爪张开位延时
AND T0038  ; 下料右夹爪张开位延时
AND T0036  ; 下料左夹爪张开位延时
OR W60.02  ; 急停带料复位触发
ANDLD
AND T0034  ; 下料提升气缸缩回位延时
AND W390.01  ; 安全门信号
SNXT(009) W405.01  ; 达复位
; rung 14
STEP(008) W405.01  ; 达复位
; rung 15: 伺服回零
LD W390.01  ; 安全门信号
SET W15.06  ; 上料机械手手动归零
SET W16.06  ; 下料机械手手动归零
SNXT(009) W405.02  ; 腔体复位
; rung 16
STEP(008) W405.02  ; 腔体复位

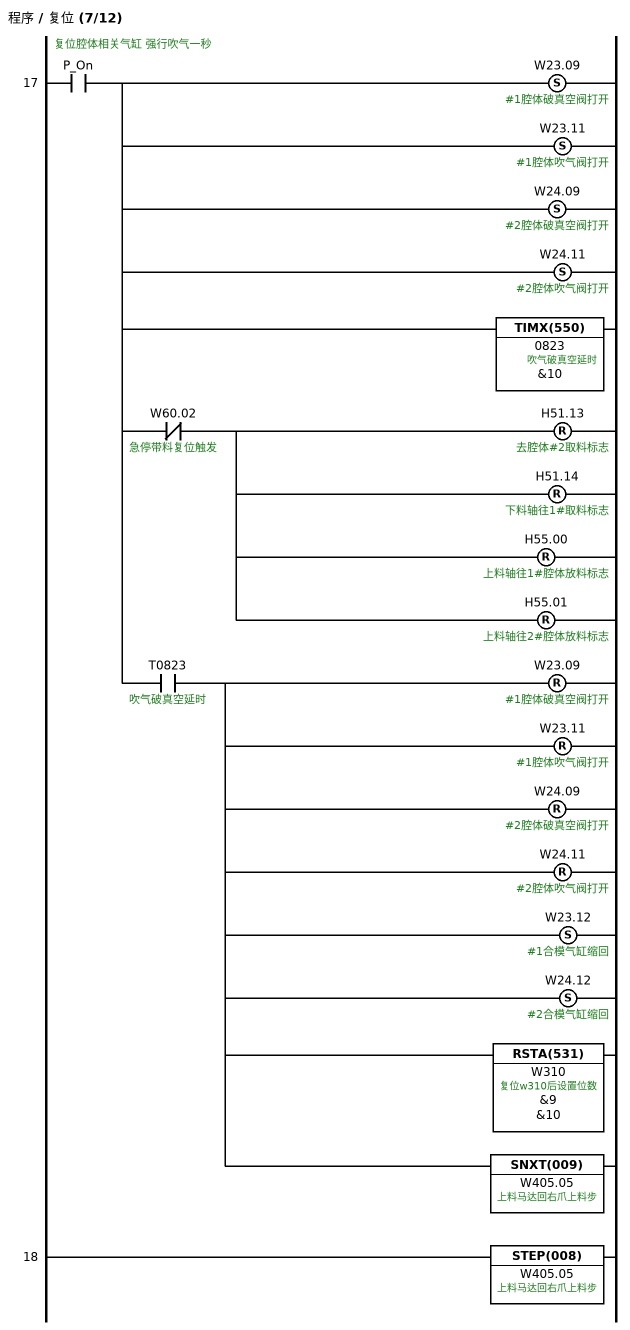
; rung 17: 复位腔体相关气缸 强行吹气一秒
LD P_On
OUT TR0
SET W23.09  ; #1腔体破真空阀打开
SET W23.11  ; #1腔体吹气阀打开
SET W24.09  ; #2腔体破真空阀打开
SET W24.11  ; #2腔体吹气阀打开
TIMX(550) 0823 &10  ; 吹气破真空延时
ANDNOT W60.02  ; 急停带料复位触发
RSET H51.13  ; 去腔体#2取料标志
RSET H51.14  ; 下料轴往1#取料标志
RSET H55.00  ; 上料轴往1#腔体放料标志
RSET H55.01  ; 上料轴往2#腔体放料标志
LD TR0
AND T0823  ; 吹气破真空延时
RSET W23.09  ; #1腔体破真空阀打开
RSET W23.11  ; #1腔体吹气阀打开
RSET W24.09  ; #2腔体破真空阀打开
RSET W24.11  ; #2腔体吹气阀打开
SET W23.12  ; #1合模气缸缩回
SET W24.12  ; #2合模气缸缩回
RSTA(531) W310 &9 &10  ; 复位w310后设置位数
SNXT(009) W405.05  ; 上料马达回右爪上料步
; rung 18
STEP(008) W405.05  ; 上料马达回右爪上料步

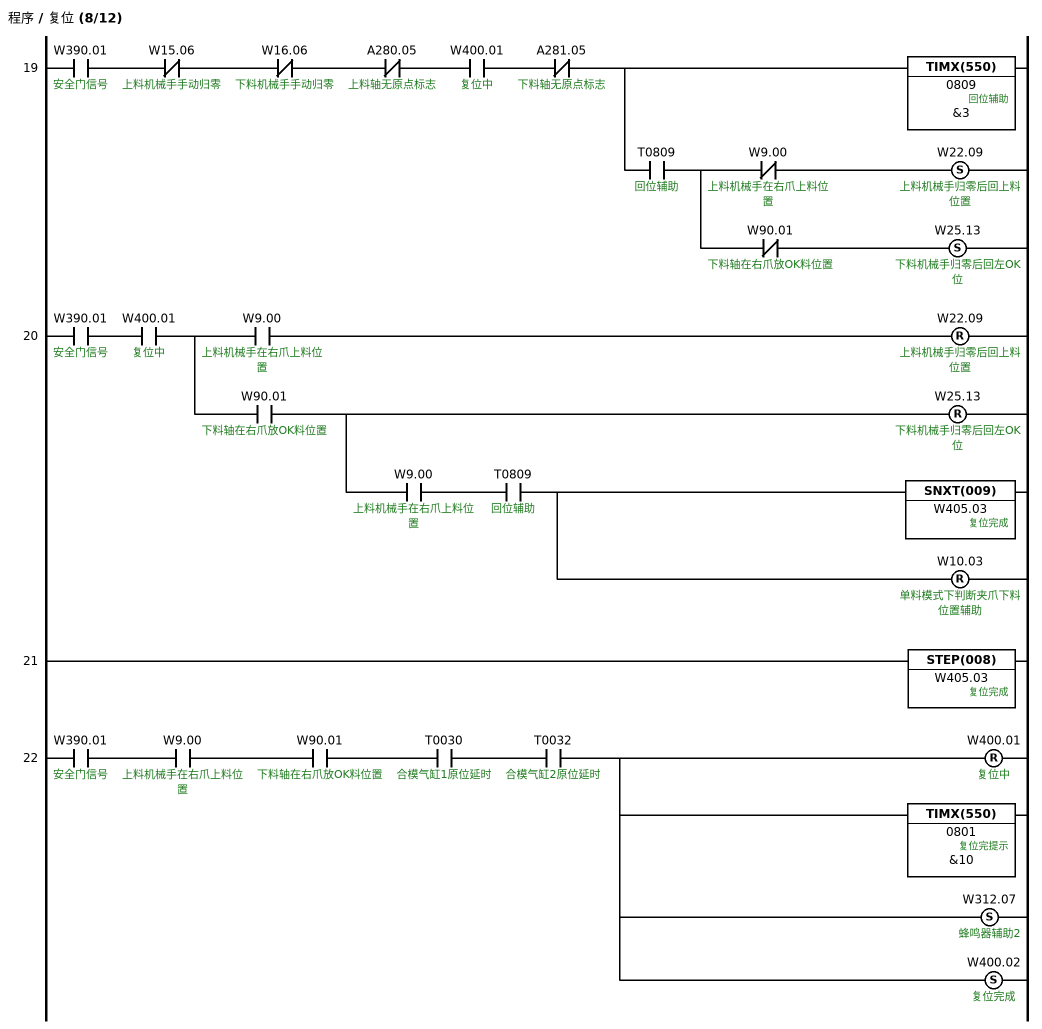
; rung 19
LD W390.01  ; 安全门信号
ANDNOT W15.06  ; 上料机械手手动归零
ANDNOT W16.06  ; 下料机械手手动归零
ANDNOT A280.05  ; 上料轴无原点标志
AND W400.01  ; 复位中
ANDNOT A281.05  ; 下料轴无原点标志
TIMX(550) 0809 &3  ; 回位辅助
AND T0809  ; 回位辅助
OUT TR0
ANDNOT W9.00  ; 上料机械手在右爪上料位置
SET W22.09  ; 上料机械手归零后回上料位置
LD TR0
ANDNOT W90.01  ; 下料轴在右爪放OK料位置
SET W25.13  ; 下料机械手归零后回左OK位
; rung 20
LD W390.01  ; 安全门信号
AND W400.01  ; 复位中
OUT TR0
AND W9.00  ; 上料机械手在右爪上料位置
RSET W22.09  ; 上料机械手归零后回上料位置
LD TR0
AND W90.01  ; 下料轴在右爪放OK料位置
RSET W25.13  ; 下料机械手归零后回左OK位
AND W9.00  ; 上料机械手在右爪上料位置
AND T0809  ; 回位辅助
SNXT(009) W405.03  ; 复位完成
RSET W10.03  ; 单料模式下判断夹爪下料位置辅助
; rung 21
STEP(008) W405.03  ; 复位完成
; rung 22
LD W390.01  ; 安全门信号
AND W9.00  ; 上料机械手在右爪上料位置
AND W90.01  ; 下料轴在右爪放OK料位置
AND T0030  ; 合模气缸1原位延时
AND T0032  ; 合模气缸2原位延时
RSET W400.01  ; 复位中
TIMX(550) 0801 &10  ; 复位完提示
SET W312.07  ; 蜂鸣器辅助2
SET W400.02  ; 复位完成

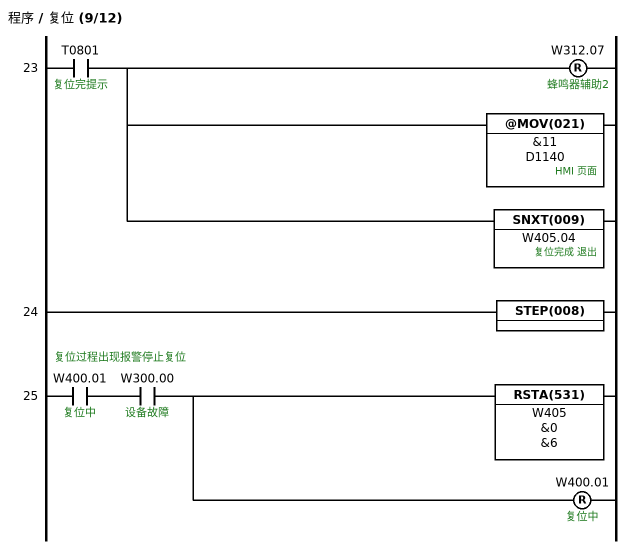
; rung 23
LD T0801  ; 复位完提示
RSET W312.07  ; 蜂鸣器辅助2
@MOV(021) &11 D1140  ; HMI 页面
SNXT(009) W405.04  ; 复位完成 退出
; rung 24
STEP(008)
; rung 25: 复位过程出现报警停止复位
LD W400.01  ; 复位中
AND W300.00  ; 设备故障
RSTA(531) W405 &0 &6
RSET W400.01  ; 复位中

